// TwinCAT 3 PLC project Pecom_Drive_Communication
// Title: DCOS PecomDriveCommunication
// Company: DCOS
// Author: DCOS
// ProjectVersion: 1.0.0
// Description: Function for Drive Communication to manroland presses replacing Baumueller Drive systems
// ProgramVersion: 3.1.4024.0
// libraries:
//   Tc2_Standard, * (Beckhoff Automation GmbH)
//   Tc2_System, * (Beckhoff Automation GmbH)
//   Tc2_TcpIp, * (Beckhoff Automation GmbH)
//   Tc2_Utilities, * (Beckhoff Automation GmbH)
// project tree:
//   DUTs/DriveInterface/ ST_DriveInterface.TcDUT, ST_DriveInterface_Ctrl.TcDUT, ST_DriveInterface_Stat.TcDUT
//   DUTs/MainAxis_Interface/ ST_MainAxisInterface_Ctrl.TcDUT, ST_MainAxisInterface_Stat.TcDUT, ST_MainAxisInterface.TcDUT
//   DUTs/Pecom_Interface/Ethernet_TCP/ NETWORK_BUFFER.TcDUT, ST_ApplicationBinaryData.TcDUT, ST_BinaryFrame.TcDUT, ST_BinaryHeader.TcDUT, ST_TCP_Puff.TcDUT
//   DUTs/Pecom_Interface/Pecom_TCP/ ST_CommunicationStatus.TcDUT, ST_Elements.TcDUT, ST_InOut_Msg.TcDUT, ST_InOut_Data.TcDUT, ST_MsgBuffer.TcDUT, ST_Restart.TcDUT, ST_Objekt.TcDUT, ST_MemberAnounce.TcDUT
//   DUTs/Pecom_Interface/Pecom_UDP/ IP_C.TcDUT, ST_UDP_Buffer.TcDUT, ST_UDP_Drive_Data.TcDUT, ST_UDP_Msg_In.TcDUT, ST_UDP_Msg_Out.TcDUT
//   DUTs/Pecom_Interface/Setup_DriveCom/ ST_SetupDriveCom.TcDUT, ST_SetupDriveComMDS.TcDUT
//   DUTs/ ST_Alarm.TcDUT, ST_TCP_Parameter.TcDUT (not stored)
//   Global Variables/Pecom_Interface/ GVL_ConnectionAlarms.TcGVL, GVL_FB.TcGVL, GVL_Pecom.TcGVL, GVL_Setup.TcGVL, TCPIP_Constants.TcGVL
//   POUs/Network Functions/TCPIP_Communication/ FB_Server.TcPOU, FB_ServerApplication.TcPOU, FB_ServerConnection.TcPOU
//   POUs/Network Functions/TCPIP_Communication/Helper POUs/ FB_FrameFifo.TcPOU, FB_LogFifo.TcPOU, F_ADSLOGHEXDATA.TcPOU
//   POUs/Network Functions/UDP_Communication/ FB_UDP_Server.TcPOU, FB_UDP_Server_RESET.TcPOU
//   POUs/Pecom Interface/ PB_Start_TCPIP.TcPOU, PB_Start_UDP.TcPOU
//   POUs/Pecom Interface/Pecom_Functions/TCP Msg Handling/ Eth_Send_Receive.TcPOU, FB_Msg_Receive.TcPOU, FB_Msg_Send.TcPOU, FB_SendReceive_TcpIp.TcPOU, Pecom_In_Out_data.TcPOU, Trigger.TcPOU
//   POUs/Pecom Interface/Pecom_Functions/ Pecom_DriveMessage.TcPOU, Pecom_Write_Alarm.TcPOU
//   POUs/Pecom Interface/Pecom_Functions/UDP Msg Handling/ FB_UDP_DriveCom.TcPOU
//   POUs/UDFB/ DWORD_OF_BYTE.TcPOU, FC_Time_To_Ramp.TcPOU, WORD_OF_BYTE.TcPOU

// ---- DUTs/DriveInterface/ST_DriveInterface.TcDUT
TYPE ST_DriveInterface :
STRUCT
	stDriveMotorInterface_stat		: ST_DriveInterface_Stat;
	stDriveMotorInterface_ctrl		: ST_DriveInterface_Ctrl;
END_STRUCT
END_TYPE

// ---- DUTs/DriveInterface/ST_DriveInterface_Ctrl.TcDUT
TYPE ST_DriveInterface_Ctrl :
STRUCT
	nSelectedMaster			:WORD;				// selected master
	nClutchedMaster			:WORD;				// clutched master
	nDriveGroup				:INT;				// Group of drives for Cutoff and Webup -> It is like the Webnumber the drive belongs to
	bReset					:BOOL;				// rising trig will reset if any fault is active
	bEnable					:BOOL;				// set to give power to motor
	bStartRun				:BOOL;				// set to start motor in slow run
	bRunRev					:BOOL;				// Direction -> set to run motor in rev direcition
	fVelocity				:LREAL;				// selected speed for slow run, if = 0 then use default vel
	fAcceleration			:LREAL;				// Acceleration in Local mode
	nGearRatio				:INT;				// For 3.Folder -> 2 or 1 ; For Paddlewheel 10000 or 20000 depends on Collect or straight!!
	// Cutoff and Speedgain
	fSyncValue				:LREAL;				// relative value to the master where motor will clutch into
	fGain					:LREAL;				// speed offset in % where such value can be used 1 = 1% faster
	
	// Positioning
	bPositionMode			:BOOL;				// POS-Mode -> set to goto a modulated positon
	bPosDirection			:BOOL;				// POS-Mode -> what direction to use when finding modulated position
	fModeModPos				:LREAL;				// POS-Mode -> selected position for modulated position 0.000 - 360.000	
	
	// 3.Folder Speed Curve
	n3Folder_Offset			:LREAL;				// 3.Folder -> Additional Cutoff offset for the 3.Folder (Fixed Value from Plc)
	n3Folder_Offset_Curve	:LREAL;				// 3.Folder -> Speed Curve Offset
	n3Folder_Degree_Curve	:LREAL;				// 3.Folder -> steepness of the speed curve
	
	// Sync Mode and Sync Speed
	bDriveSyncMode_FW		:BOOL;				// Sync Forward --> Syncronisation-Speed can be any speed 
	bDriveSyncMode_BW		:BOOL;				// Sync Backward --> Syncronisation-Speed must be < Machine speed exept N= 0 !!!
	bDriveSyncMode_SW		:BOOL;				// Sync Shortest way --> Syncronisation-Speed must be < Machine speed exept N= 0 !!!
	fSyncSpeed				:LREAL;				// set to desired sync offset speed Degree/sec for sync to Main Axis
	fSpeedCR_Permill		:LREAL;				// For PU only!! -> 100.0000 Promill OR 0.0400 Promill
	fSpeedCR_DegreeS		:LREAL;				// For Folder only!! -> 20,0000 Degree/sec OR 1,0000 Degree/sec
	fSpeedCutoff_Permill_Vari	:LREAL;				// set to desired sync offset speed Promill -> eg. 100.0000 Promill OR 0.2800 Promill
	fSpeedCutoff_Degree		:LREAL;				// set to desired sync offset speed Degree/sec 
	
	
	// Webtension Control Mode 
	nWebTc_Mode				:INT;				// WebTc	-> 11=off, 12=On  , 13=Tempor. Off
	fWebTc_SpeedGain		:LREAL;				// WebTc	-> Speedgain in manual mode in permill * 100 (eg 0.01‰ * 100)
	fWebTc_WebTension		:LREAL;				// WebTc	-> Webtension in N In Automode
	
	// something ??
	nSwitchPararmeter		:DINT;				// Switches between 2 parameter sets -> 0 or 1
	bDriveMode				:BOOL;				// 11 = position Ctrl, 13 = speed Ctrl, 14 = Tourque slave
END_STRUCT
END_TYPE

// ---- DUTs/DriveInterface/ST_DriveInterface_Stat.TcDUT
TYPE ST_DriveInterface_Stat :
STRUCT
	bEnabled			:BOOL;			// drive is under power
	
	fActVel				:LREAL;			// acutal vel, untis/s
	fActTorque			:LREAL;			// Actual Torque in %
	fTemp				:REAL;			// actual motor temp
	fI2T				:REAL;			// actual current overload accumulator in % when at 100% drive will trip  
	
	bZeroSpeed			:BOOL;			// motor at zerospeed (standstill)
	
	// Sync Feedback
	bInSync				:BOOL;			// Drive is in Sync with master Axis
	
	// Error Handling
	bError				:BOOL;			// has fault	
	nErrorCode			:DINT;			// error code	
	
	//Positioning Mode
    bAtModPos			:BOOL;			// set when in modulated position mode and at required pos	
	fActPos				:LREAL;			// actual modulated position, units
	fSyncPosDifference	:LREAL;			// Difference of the MainAxis to the local Position
	// Webtension Control Mode 
	fWebTc_SpeedGain	:LREAL;		// WebTc	-> Speedgain in manual mode in permill * 100 (eg 0.01‰ * 100)
	fWebTc_WebTension	:LREAL;		// WebTc	-> Webtension in N In Automode
	
	
	// divers
	bCoolingFanStarted	:BOOL;			// coolingfan running
	bBrakeReleased		:BOOL;			// breake is off
END_STRUCT
END_TYPE

// ---- DUTs/MainAxis_Interface/ST_MainAxisInterface_Ctrl.TcDUT
TYPE ST_MainAxisInterface_Ctrl :
STRUCT
	bReset					:BOOL;						// rising trig will reset if any fault is active
	
	bEnable					:BOOL;						// set to give power to motor
	bStartRun				:BOOL;						// set to start motor in slow run
	fVelocity				:LREAL;						// selected speed for slow run, if = 0 then use default vel
	fAcceleration			:LREAL;						// Acceleration in Local mode
	
	// Cutoff and Speedgain
	fCutoffValue			:ARRAY[0..31] OF LREAL;		// Cutoff for each DriveGroup (equals the web number )
	
	// Aray of Cutoff values for each group
	aGroup_Cutoff			:	ARRAY[0..15] OF LREAL;	// Cutoff from SKS for each web Group
	
	// Each Bit represents a group which is doing a webbing up. Only drives in this group are turning
	aGroup_WebUpDrives		:	ARRAY[0..15] OF BOOL;	// Group which is involved in a webup			
	
END_STRUCT
END_TYPE

// ---- DUTs/MainAxis_Interface/ST_MainAxisInterface_Stat.TcDUT
TYPE ST_MainAxisInterface_Stat :
STRUCT
	bEnabled			:BOOL;			// drive is under power
	
	fActVel				:LREAL;			// acutal vel, untis/s
	
	fActPos				:LREAL;			// actual modulated position, units
	
	// P1160 Sync Feedback for each Drive Group (Bit 0 = Group 0 and so on)
	bInSync				:WORD;			// Status of the Sync Position for each DRIVE-GROUP (Is a drive in a group not in sync -> BIT is High)
	
	bZeroSpeed			:BOOL;			// motor at zerospeed (standstill)
	
	// Error Handling
	bError				:BOOL;			// Main Axis has a fault	


END_STRUCT
END_TYPE

// ---- DUTs/MainAxis_Interface/ST_MainAxisInterface.TcDUT
TYPE ST_MainAxisInterface :
STRUCT
	stMainAxisInterface_stat		: ST_MainAxisInterface_Stat;
	stMainAxisInterface_ctrl		: ST_MainAxisInterface_Ctrl;
END_STRUCT
END_TYPE

// ---- DUTs/Pecom_Interface/Ethernet_TCP/NETWORK_BUFFER.TcDUT
TYPE NETWORK_BUFFER :
STRUCT
	SIZE : UINT;
	BUFFER : ARRAY[0..Pecom_TCP_Puffer_Size] OF BYTE;
END_STRUCT
END_TYPE

// ---- DUTs/Pecom_Interface/Ethernet_TCP/ST_ApplicationBinaryData.TcDUT
(* Simple binary user data (8 byte aligned) *)
TYPE ST_ApplicationBinaryData :
STRUCT
	aData		: ARRAY[0..Pecom_TCP_Puffer_Size] OF BYTE; // 700 Byte
	reserved	: ARRAY[0..2] OF BYTE;(* Alignment data: 3 byte *)

END_STRUCT
END_TYPE

// ---- DUTs/Pecom_Interface/Ethernet_TCP/ST_BinaryFrame.TcDUT
(* Simple binary TCP/IP frame (8 byte aligned) *)
TYPE ST_BinaryFrame :
STRUCT
//	head	: ST_BinaryHeader;(* Frame header (16 byte) *)
	data 	: ST_ApplicationBinaryData;(* User data (120 byte) *)

	(* Total frame size = 136 byte *)
END_STRUCT
END_TYPE

// ---- DUTs/Pecom_Interface/Ethernet_TCP/ST_BinaryHeader.TcDUT
(* Simple binary TCP/IP frame header (8 byte aligned) *)
TYPE ST_BinaryHeader :
STRUCT
	dwStart		: DWORD	:= 16#BECF1234;	(* Start bytes *)
	cbLength	: UDINT(0..PLCPRJ_BUFFER_SIZE) := 0;(* Max. length of attached binary data *)
	nS			: UDINT := 0;(* Send counter *)
	nR			: UDINT	:= 0;(* Receive counter *)
	
	(* Total header data size = 16 byte *)
END_STRUCT
END_TYPE

// ---- DUTs/Pecom_Interface/Ethernet_TCP/ST_TCP_Puff.TcDUT
TYPE ST_TCP_Puff:
STRUCT
	Conected	: BOOL;
	Ip_Adresss	: T_IPv4addr;
	PecomTNR  	: INT;		 
	R_Buf		: NETWORK_BUFFER;
	S_Buf		: NETWORK_BUFFER;
END_STRUCT
END_TYPE

// ---- DUTs/Pecom_Interface/Pecom_TCP/ST_CommunicationStatus.TcDUT
TYPE ST_CommunicationStatus :
STRUCT
	stRestart				:	ST_Restart;
	bTCP_Connect			:	ARRAY[0..NR_OF_DRIVEMASTERS] OF BOOL;
	bUDP_Connect			:	ARRAY[0..NR_OF_DRIVEMASTERS] OF BOOL;
END_STRUCT
END_TYPE

// ---- DUTs/Pecom_Interface/Pecom_TCP/ST_Elements.TcDUT
TYPE ST_Elements :
STRUCT
	Nummer	  : INT;	(* Gegenstelle*)
	KNG	   	  : INT;
	ANFTYP	  : INT;
	SNSTIV	  : INT;
	ZYKTME	  : INT;
	MASEIN	  : INT;
	flag	  : BOOL;
END_STRUCT
END_TYPE

// ---- DUTs/Pecom_Interface/Pecom_TCP/ST_InOut_Msg.TcDUT
TYPE ST_InOut_Msg :
STRUCT
	number_of_buffers	:	INT;
	buffer_overfow		:	BOOL;
	Pecom_Tnr			:	ARRAY [1..40] OF INT;
	valid				:	ARRAY [1..40] OF BOOL;
	stMsgBuffer			:	ARRAY [1..40] OF  ST_MsgBuffer;	// 40 x 950 Words Buffer
END_STRUCT

END_TYPE

// ---- DUTs/Pecom_Interface/Pecom_TCP/ST_InOut_Data.TcDUT
TYPE ST_InOut_Data :
STRUCT
	Error						: SINT;
	Hand_Shake					: SINT;
    Receiver  					: INT;
	Sender     					: INT;
	Typ		 					: INT;
	NFB		  					: INT;
	Lg_Byte	 					: INT;
	KDO							: INT;
   	data						: ARRAY[7..950] OF INT;
	data_Max  					: INT;
   	BLK_Pointer 				: INT;
	DSK_Pointer 				: INT;
	nNumber_of_messages			: INT;
	nNumber_of_Error			: INT;
	nUnknown_message			: INT;
    data_transfer_ready     	: BOOL;
	data_are_valid				: BOOL;
	Send_data					: BOOL;
    job_running             	: BOOL;
	job_done 					: BOOL;
	job_not_done  				: BOOL;
	job_timeout					: BOOL;
	Release_first_value			: BOOL;
END_STRUCT
END_TYPE

// ---- DUTs/Pecom_Interface/Pecom_TCP/ST_MsgBuffer.TcDUT
(* Ethernetpuffer *)
TYPE ST_MsgBuffer :
STRUCT
	MSG	: ARRAY [0..950] OF	 WORD;	// Ethernetpuffer 950 Words
END_STRUCT
END_TYPE

// ---- DUTs/Pecom_Interface/Pecom_TCP/ST_Restart.TcDUT
TYPE ST_Restart :
STRUCT
	akt							: BOOL;
	TLN							: ARRAY[1..4]	OF	INT;
END_STRUCT
END_TYPE

// ---- DUTs/Pecom_Interface/Pecom_TCP/ST_Objekt.TcDUT
TYPE ST_Objekt :
STRUCT
    OBJART	  		: INT;
	OBJLGE	  		: INT;
	OBJGRP	  		: INT;
	OBJEIN	  		: INT;
	OBJLFN	  		: INT;
    AUFTRAG	  		: INT;
	KOM_RCK   		: BOOL;
	AKTIV			: BOOL;
	TLN				: ARRAY [0..4] OF ST_Elements;
	Read_Data 		: BOOL;
	Send_Data 		: BOOL;
	In_data			: ARRAY [0..400] OF INT;
	Out_data		: ARRAY [0..400] OF INT;

END_STRUCT
END_TYPE

// ---- DUTs/Pecom_Interface/Pecom_TCP/ST_MemberAnounce.TcDUT
TYPE ST_MemberAnounce :
STRUCT
	Laenge		:	WORD;
	receiver	:	WORD;
	Sender		:	WORD;
	Typ			:	WORD;
	Reserve		:	WORD;
	N_Laenge	:	WORD;
	Kommando	:	WORD;
END_STRUCT

END_TYPE

// ---- DUTs/Pecom_Interface/Pecom_UDP/IP_C.TcDUT
TYPE IP_C :
STRUCT
	C_PORT : WORD;						(*W Portnummer                                               *)
	C_IP : DWORD;						(*W IP-Adresse gepackt wwxxyyzz = www.xxx.yyy.zzz            *)
	C_STATE : BYTE;						(*R Verbindungsstatus ON/OFF + Flanke ON/OFF                 *)
	C_ENABLE : BOOL;					(*W Freigabe für Connect                                     *)
	R_OBSERVE : BOOL;					(*W Empfang ueberwachen                                      *)
	TIME_RESET : BOOL;					(*W Alle Timer ruecksetzen                                   *)
	ERROR : DWORD;					    (*R vvwwxxyy (vv = CON_ERROR, ww = SEN_ERROR, xx = REC_ERROR *)
	MAILBOX : ARRAY [1..16] OF BYTE;	(*I Mailbox: Datenbereich für Bausteindatenaustausch         *)
END_STRUCT
END_TYPE

// ---- DUTs/Pecom_Interface/Pecom_UDP/ST_UDP_Buffer.TcDUT
TYPE ST_UDP_Buffer :
STRUCT	
	Ip_Adresss		: T_IPv4addr;
	nDriveMemberNr	: INT;
	nPLCMemberNr	: INT;
	SIZE 			: UINT;
	BUFFER 			: ARRAY[0..Pecom_TCP_Puffer_Size] OF BYTE;
END_STRUCT
END_TYPE

// ---- DUTs/Pecom_Interface/Pecom_UDP/ST_UDP_Drive_Data.TcDUT
TYPE ST_UDP_Drive_Data :
	STRUCT
		sRemote_IP_Adress		: T_IPv4Addr;
		nDriveMemberNr			: INT;			// Own Pecom Member Nr. (Old MDS Pecom Nr)
		nPLCMemberNr			: INT;			// PLC Pecom Member Nr.
		bConnectionState		: BOOL;
		aDriveData_In			: ARRAY[0..50] OF ST_UDP_Msg_In;
		aDriveData_Out			: ARRAY[0..50] OF ST_UDP_Msg_Out;
	END_STRUCT
END_TYPE

// ---- DUTs/Pecom_Interface/Pecom_UDP/ST_UDP_Msg_In.TcDUT
TYPE ST_UDP_Msg_In :
	STRUCT
		nDriveSercos_Id			:	INT;
		nControlword			:	WORD;
		nSetpoint_speed			:	INT;	// Speed in Rev/10
		nSetpoint_Acceleration	:	INT;	// Acceleration /10 (Time in relation to Vmax eg. 37500 rev/h)
		bHandShake				:	BOOL;	// UDP Bit 0 Handshake
		bSyncRunMode			:	BOOL;	// UDP Bit 8 Syncron Run Operating Mode
		bPositionMode			:	BOOL;	// UDP Bit 9 Positioning Operating Mode
		bDriveEnable			:	BOOL;	// UDP Bit 14 Drive Enable
		bDriveStop				:	BOOL;	// UDP Bit 15 Drive Stop -> Drive is locked
	END_STRUCT
END_TYPE

// ---- DUTs/Pecom_Interface/Pecom_UDP/ST_UDP_Msg_Out.TcDUT
TYPE ST_UDP_Msg_Out :
	STRUCT
		nDriveSercos_Id			:	INT;
		nStatusWord				:	WORD;
		nActual_speed			:	INT;	// Actual Speed in Rev/10
		nActual_torque			:	INT;	// Torque in %
		bHandShake				:	BOOL;	// UDP Bit 0 Handshake
		bInSync					:	BOOL;	// UDP Bit 6 Drive in Sync
		bCommandDone			:	BOOL;	// UDP Bit 7 the last Command is executed
		bDriveFault				:	BOOL;	// UDP Bit 13 Drive has a fault
		bDriveActive			:	BOOL;	// UDP Bit 14 Drive is active (Enabled and run)
		bDriveReady				:	BOOL;	// UDP Bit 15 Drive is ready
	END_STRUCT
END_TYPE

// ---- DUTs/Pecom_Interface/Setup_DriveCom/ST_SetupDriveCom.TcDUT
TYPE ST_SetupDriveCom :
	STRUCT
		nDriveNumber			: INT;			// MDxx -> Drive number in the drive array and the Axis
		sDriveName				: STRING;		// Label of the drive eg. in the drawings
		sDriveDescription		: STRING;		// Description or function of the drive	in the press	
		sLocalIP				: STRING;		// Own Ip adress (Socket) where the Pecom send the Messages to
		sRemoteIP				: STRING;		// Ip adress of the pecom Partner-plc system 
		nDriveMemberNr			: INT;
		nPLCMemberNr			: INT;
        nSercosID               : INT;			// Indicate the position of the drive in the UDP-Msg Stack
	END_STRUCT
END_TYPE

// ---- DUTs/Pecom_Interface/Setup_DriveCom/ST_SetupDriveComMDS.TcDUT
TYPE ST_SetupDriveComMDS :
	STRUCT
		nUnitNr					: INT;
		stSetup_MDS_IP			: T_IPv4addr;
		nPLCMemberNr_1			: INT;
		nPLCMemberNr_2			: INT;
		nDriveMemberNr			: INT;
	END_STRUCT
END_TYPE

// ---- DUTs/ST_Alarm.TcDUT
TYPE ST_Alarm :
STRUCT
		Status				:	BOOL;
		ernr				:	INT;
		objektnr			:	INT;
		ort1				:	INT;
		ort2				:	INT;
		ort3				:	INT;
		ort4				:	INT;
		ort5				:	INT;
		ort6				:	INT;
		ort7				:	INT;
		ort8				:	INT;
		quitt				:	INT;
		sperre				:	INT;
		gruppe				:	INT;
END_STRUCT
END_TYPE

// ---- Global Variables/Pecom_Interface/GVL_ConnectionAlarms.TcGVL
VAR_GLOBAL
	bAlarm_NoUDP_Connection		:	ARRAY[0..NR_OF_DRIVEMASTERS] OF BOOL;
	bAlarm_NoTCP_Connection		:	ARRAY[0..NR_OF_DRIVEMASTERS] OF BOOL;

END_VAR

// ---- Global Variables/Pecom_Interface/GVL_FB.TcGVL
VAR_GLOBAL
	FB_UDP_Connection_arr	: ARRAY[0..NR_OF_DRIVEMASTERS] OF FB_UDP_DriveCom;
END_VAR

// ---- Global Variables/Pecom_Interface/GVL_Pecom.TcGVL
VAR_GLOBAL
	
	stDrive_Data_arr		:	ARRAY[0..NR_OF_DRIVEMASTERS]	OF ST_UDP_Drive_Data;
	aTcpPuff				:   ARRAY[0..NR_OF_DRIVEMASTERS] 	OF ST_TCP_Puff;
	UDP_SERVER_RESET 		: 	BYTE; 			// Set to 0 to close and reopen the UPD Socket (use R_TRIG !!) OK-State is 2
	
	stComStatus				:	ST_CommunicationStatus;
	(* PECOM messages *)
	st_IN_PecomMsg			:	ST_InOut_Msg;		// The TCP IN Buffer "R_BUF_A.BUFFER[x]" is copied into this Buffer
	st_OUT_PecomMsg			:	ST_InOut_Msg;		// This Buffer is transfered into the TCP Out Buffer -> "S_BUF_A.BUFFER[x]"
	st_IN_Objects			:	ST_InOut_Data;		// "st_IN_PecomMsg" are sorted into st_IN_Objects
	st_OUT_Objects			:	ST_InOut_Data;		// single "st_OUT_Objects" are sorted into "st_OUT_Objects_Buffer" and this finally into "st_OUT_PecomMsg"
	st_OUT_Objects_Buffer	:	ST_InOut_Data;		// "st_OUT_Objects_Buffer" transfered into "st_OUT_PecomMsg"
	st_OUT_Alarms			:	ST_InOut_Data;		// struct for Alarm Messages
	st_OUT_Alarms_Buffer	:	ST_InOut_Data;		// struct Buffer for Alarm Messages

END_VAR

// ---- Global Variables/Pecom_Interface/GVL_Setup.TcGVL
VAR_GLOBAL	
	stSetup_MdsCom				: ARRAY [0..NR_OF_DRIVEMASTERS] OF ST_SetupDriveComMDS;		
	stSetup_DriveCom			: ARRAY [0..50] 				OF ST_SetupDriveCom;
END_VAR

// ---- Global Variables/Pecom_Interface/TCPIP_Constants.TcGVL
VAR_GLOBAL CONSTANT
	
	NR_OF_DRIVEMASTERS						: USINT	:= 11;		(* Max. Number of TCP Connection and Server Instances *)

	Pecom_TCP_Puffer_Size					: INT	:= 700;	(* Puffer for the Pecom In/Out Messages *)
	PLCPRJ_BUFFER_SIZE						: UDINT := 1000;(* Max. internal fifo/receiver buffer size *)

(*	PLCPRJ_CLIENT_SEND_CYCLE_TIME			: TIME := T#1S; not used at server side *)
	PLCPRJ_RECEIVE_POLLING_TIME				: TIME := T#100MS;
	PLCPRJ_RECEIVE_TIMEOUT					: TIME := T#50S;

	(* Some project specific error codes *)
	PLCPRJ_ERROR_RECEIVE_TIMEOUT			: UDINT := 16#8101;(* Receive timeout *)
	PLCPRJ_ERROR_SENDFIFO_OVERFLOW			: UDINT := 16#8102;(* Send fifo overflow *)
	PLCPRJ_ERROR_RECFIFO_OVERFLOW			: UDINT := 16#8103;(* Receive fifo overflow *)
	PLCPRJ_ERROR_INVALID_FRAME_FORMAT		: UDINT := 16#8104;(* Invalid frame format/data *)
	
END_VAR

// ---- POUs/Pecom Interface/Pecom_Functions/UDP Msg Handling/FB_UDP_DriveCom.TcPOU
FUNCTION_BLOCK FB_UDP_DriveCom
VAR_INPUT
	sRemote_IP			: T_IPv4Addr;
	nDriveMemberNr		: INT;			// Own Pecom Member Nr. (Old MDS Nr)
	nPLCMemberNr		: INT;			// PLC Pecom Member Nr.
	p_UDP_DriveData		: POINTER TO ST_UDP_Drive_Data;
	S_BUF				: POINTER TO ST_UDP_Buffer;		// UDP Send Buffer It is hand over to the UDP Socket 
	R_BUF				: POINTER TO ST_UDP_Buffer;		// UDP Receive Buffer It comes from the UDP Socket 	

END_VAR
VAR_OUTPUT
	bAlarmNoConnection	: BOOL;
END_VAR

VAR
	nInPackageCount			: INT;
	bTimeout				: BOOL;
	TON_Timeout				: TON;
	nStackPointer			: INT;
	nDriveNumber			: INT;
	
	TO_PECOM				: ARRAY[0..650]	OF	WORD;
	TO_PECOM_old			: ARRAY[0..650]	OF	WORD;
	
	
	bSendRequest			: BOOL;
	nMsgSize				: INT;
	p						: INT;
	i						: INT;
	k						: UINT;
	sIPTEST: STRING(15);
END_VAR

(************************************************************************************************)
(*****				 					Ethernet UDP 										*****)
(***** UDP Communication between the PLC <--> Drive System 									*****)
(***** 																						*****)
(************************************************************************************************)
(*****			Time out or no connection after 7s of no Message		*****)
//Set the Timeout for connection control
bTimeout	:=	TRUE;
// Reset the TimeOut when you received a valid UDP-package
IF (R_BUF^.SIZE > 0 AND R_BUF^.Ip_Adresss = sRemote_IP) 
THEN
	bTimeout := FALSE;	
	nInPackageCount	:=	nInPackageCount	+	1;		// Diagnose Only!!
	sIPTEST	:= R_BUF^.Ip_Adresss;
END_IF
TON_Timeout(IN:= bTimeout, PT:=T#6S);
bAlarmNoConnection	:=	TON_Timeout.Q;

// Connection Flag in the UDP Buffer
p_UDP_DriveData^.bConnectionState := NOT bAlarmNoConnection	;

(****************************************************************************************)
(***							Receive Messages									*****)
(* If In-Buffer size is gt the 0 transfer the content to the  p_DriveData array			*)
(* In 1 Msg can be max. 48 drives controlled. Each on is identified by its Sercos-Id	*)
(****************************************************************************************)

IF		(R_BUF^.SIZE > 0 AND R_BUF^.Ip_Adresss = sRemote_IP)
THEN	
	p_UDP_DriveData^.sRemote_IP_Adress	:= 	sRemote_IP;
	p_UDP_DriveData^.nDriveMemberNr		:=	R_BUF^.nDriveMemberNr;	
	p_UDP_DriveData^.nPLCMemberNr		:=	R_BUF^.nPLCMemberNr;
	nStackPointer	:=	26;	// Pointer offset to the First drive information in the Msg
	
	FOR nDriveNumber	:= 0 TO 48
				DO
					p_UDP_DriveData^.aDriveData_In[nDriveNumber].nDriveSercos_Id		:=	WORD_TO_INT(WORD_OF_BYTE(R_BUF^.BUFFER[nStackPointer+1],R_BUF^.BUFFER[nStackPointer]));
					p_UDP_DriveData^.aDriveData_In[nDriveNumber].nControlword 			:=	WORD_OF_BYTE(R_BUF^.BUFFER[nStackPointer+2],R_BUF^.BUFFER[nStackPointer+3]);
					p_UDP_DriveData^.aDriveData_In[nDriveNumber].nSetpoint_speed 		:=	WORD_TO_INT(WORD_OF_BYTE(R_BUF^.BUFFER[nStackPointer+4],R_BUF^.BUFFER[nStackPointer+5]));
					p_UDP_DriveData^.aDriveData_In[nDriveNumber].nSetpoint_Acceleration :=	WORD_TO_INT(WORD_OF_BYTE(R_BUF^.BUFFER[nStackPointer+6],R_BUF^.BUFFER[nStackPointer+7]));
					
					// Assign the Control bits
					p_UDP_DriveData^.aDriveData_In[nDriveNumber].bHandShake				:=	p_UDP_DriveData^.aDriveData_In[nDriveNumber].nControlword.0;
					p_UDP_DriveData^.aDriveData_In[nDriveNumber].bSyncRunMode			:=	p_UDP_DriveData^.aDriveData_In[nDriveNumber].nControlword.8;
					p_UDP_DriveData^.aDriveData_In[nDriveNumber].bPositionMode			:=	p_UDP_DriveData^.aDriveData_In[nDriveNumber].nControlword.9;
					p_UDP_DriveData^.aDriveData_In[nDriveNumber].bDriveEnable			:=	p_UDP_DriveData^.aDriveData_In[nDriveNumber].nControlword.14;
					p_UDP_DriveData^.aDriveData_In[nDriveNumber].bDriveStop				:=	p_UDP_DriveData^.aDriveData_In[nDriveNumber].nControlword.15;

					nStackPointer	:= nStackPointer +12;
	END_FOR;		
END_IF

(****************************************************************************************)
(***							Send Messages									*****)
(* If In-Buffer size is gt the 0 transfer the content to the  p_DriveData array			*)
(* In 1 Msg can be max. 48 drives controlled. Each on is identified by its Sercos-Id	*)
(****************************************************************************************)
TO_PECOM_old := TO_PECOM;
(*****************************************************)
(** Build the Header of the Message					**)
(**	static part of the message 						**)
(*****************************************************)

TO_PECOM[0]		:=	INT_TO_WORD(nPLCMemberNr);
TO_PECOM[1]		:=	INT_TO_WORD(nDriveMemberNr);
TO_PECOM[2]		:=	WORD#153;
TO_PECOM[3]		:=	WORD#0;
TO_PECOM[4]		:=	WORD#600;	(* 12 Byte x 49 Drives *)
TO_PECOM[5]		:=	WORD#10912;	(* Message Type	*)
TO_PECOM[6]		:=	WORD#0;
TO_PECOM[7]		:=	WORD#1;
TO_PECOM[8]		:=	WORD#302;	(* OBJART *)
TO_PECOM[9]		:=	WORD#49;	(* number of drives *)
TO_PECOM[10]	:=	WORD#12;	(* OBJLGE per Drive in Byte*)


(*****************************************************)
(**	dynamic part of the message 					**)
(*****************************************************)
// Write the Drive struct into the temp. Send-Buffer
p	:=	11;
	FOR nDriveNumber	:= 0 TO 48
		DO	p_UDP_DriveData^.aDriveData_Out[nDriveNumber].nStatusWord	:= 0;	// Clear the Status
		
			// reply to the UDP Handshake Bit
			p_UDP_DriveData^.aDriveData_Out[nDriveNumber].bHandShake		:= p_UDP_DriveData^.aDriveData_In[nDriveNumber].bHandShake;

			// Write the Status word
			p_UDP_DriveData^.aDriveData_Out[nDriveNumber].nStatusWord.0		:= p_UDP_DriveData^.aDriveData_Out[nDriveNumber].bHandShake;
			p_UDP_DriveData^.aDriveData_Out[nDriveNumber].nStatusWord.6		:= p_UDP_DriveData^.aDriveData_Out[nDriveNumber].bInSync;
			p_UDP_DriveData^.aDriveData_Out[nDriveNumber].nStatusWord.7		:= p_UDP_DriveData^.aDriveData_Out[nDriveNumber].bCommandDone;
			p_UDP_DriveData^.aDriveData_Out[nDriveNumber].nStatusWord.13	:= p_UDP_DriveData^.aDriveData_Out[nDriveNumber].bDriveFault;			
			p_UDP_DriveData^.aDriveData_Out[nDriveNumber].nStatusWord.14	:= p_UDP_DriveData^.aDriveData_Out[nDriveNumber].bDriveReady;
			p_UDP_DriveData^.aDriveData_Out[nDriveNumber].nStatusWord.15	:= p_UDP_DriveData^.aDriveData_Out[nDriveNumber].bDriveActive;
		
			TO_PECOM[p]		:=	2056;
			TO_PECOM[p+1]	:=	1;
			TO_PECOM[p+2]	:=	ROR(INT_TO_WORD(p_UDP_DriveData^.aDriveData_In[nDriveNumber].nDriveSercos_Id),8);
			TO_PECOM[p+3]	:=	p_UDP_DriveData^.aDriveData_Out[nDriveNumber].nStatusWord;
			TO_PECOM[p+4]	:=	INT_TO_WORD(p_UDP_DriveData^.aDriveData_Out[nDriveNumber].nActual_speed);
			TO_PECOM[p+5]	:=	INT_TO_WORD(p_UDP_DriveData^.aDriveData_Out[nDriveNumber].nActual_torque);
			nMsgSize		:=  p *2;
			p	:= p + 6;
			
END_FOR

(*****************************************************)
(***	Create a send request					******)
(*****************************************************)
// Compare old and new State and create a SendRequest

IF 	MEMCMP(ADR(TO_PECOM), ADR(TO_PECOM_old), SIZEOF(TO_PECOM_old)) <> 0	
	OR	(R_BUF^.SIZE > UINT#0 AND R_BUF^.Ip_Adresss = sRemote_IP)		(*message was incoming and must be replied*)
THEN
	bSendRequest:=	TRUE;
END_IF

(*****************************************************)
(* send the message to the remote plc*)
(*****************************************************)
IF bSendRequest THEN	
	IF	S_BUF^.SIZE	=	UINT#0 (* last message was done *)
	THEN
		k	:=	0;
		FOR	i	:= 0 TO nMsgSize
			DO
				S_BUF^.BUFFER[k]		:=	WORD_TO_BYTE(SHR(TO_PECOM[i],8));
				k	:=	k + 1;
				S_BUF^.BUFFER[k]		:=	WORD_TO_BYTE(TO_PECOM[i]);				
				k	:=	k + 1;
			END_FOR;
		S_BUF^.Ip_Adresss 				:= sRemote_IP;
		S_BUF^.nPLCMemberNr				:= nPLCMemberNr;
		S_BUF^.nDriveMemberNr			:= nDriveMemberNr;
		S_BUF^.SIZE						:= k;			(* send it *)
		bSendRequest 					:= FALSE;		
	END_IF;	
END_IF

(********************************************************)
(* Reset the Receiving buffer and wait for next message	*)
(*****************************************************)
IF R_BUF^.Ip_Adresss = sRemote_IP THEN
	R_BUF^.SIZE	:=	0;
	R_BUF^.Ip_Adresss := '';
END_IF

END_FUNCTION_BLOCK

// ---- POUs/UDFB/WORD_OF_BYTE.TcPOU
FUNCTION WORD_OF_BYTE : WORD
VAR_INPUT
	B1 : BYTE;
	B0 : BYTE;
END_VAR


(*
version 1.4	18. jul. 2009
programmer 	hugo
tested by		tobias

this function creates a word from 2 individual bytes

*)

WORD_OF_BYTE := SHL(BYTE_TO_WORD(B1),8) OR BYTE_TO_WORD(B0);

(* revision history
hm	24. jan 2007	rev 1.0
	original version

hm	2. jan 2008	rev 1.1
	improved performance

hm	19. feb 2008	rev 1.2
	replaced and with or for better compatibility

hm	23. apr. 2008	rev 1.3
	reverse order of inputs to be more logical

hm	18. jul. 2009	rev 1.4
	added type conversions for compatibility reasons

*)

END_FUNCTION

// ---- POUs/Network Functions/TCPIP_Communication/FB_Server.TcPOU
FUNCTION_BLOCK FB_Server
VAR_IN_OUT
	hServer			: T_HSERVER;(* Server connection handle *)
END_VAR
VAR_INPUT
	nServer_Id		: INT;
	sSrvNetID		: T_AmsNetID	:= '';(* TwinCAT TCP/IP server network address *)
	bEnable			: BOOL 			:= FALSE;(* TRUE => Enable server data exchange, FALSE => Disable *)
	bLog			: BOOL 			:= FALSE;(* TRUE => Enable log message output, FALSE => Disable *)
	sPrefix			: STRING 		:= 'SERVER::';(* Log message description string (allows the identification of log message source) *)
END_VAR
VAR_OUTPUT
	eState			: E_SocketConnectionState := eSOCKET_DISCONNECTED;(* TCP/IP connection state *)
END_VAR
VAR
	fbApplication 	: FB_ServerApplication;(* Server application control function block *)
	fbConnection	: FB_ServerConnection;(* Server data exchange control function block *)
	fbTx 			: FB_FrameFifo;(* Tx fifo *)
	fbRx 			: FB_FrameFifo;(* Rx fifo *)
	fbLog			: FB_LogFifo;(* Log/debug/error fifo *)
END_VAR

(*-------------------------- Trigger data exchange -----------------------------------------------*)
fbConnection( 	hServer := hServer, sSrvNetID := sSrvNetID, 
				fbRx := fbRx, fbTx := fbTx, fbLog := fbLog, 
				bEnable := bEnable, bLog := bLog, sPrefix := sPrefix, eState=>eState );
	
IF fbConnection.eState = eSOCKET_CONNECTED THEN(* Connection established *)
	aTcpPuff[nServer_Id].Conected := TRUE;
	aTcpPuff[nServer_Id].Ip_Adresss := fbConnection.sIpAdress;
	fbApplication( fbTx := fbTx, fbRx := fbRx, fbLog := fbLog, nServer_Id := nServer_Id );
ELSE	
	aTcpPuff[nServer_Id].Ip_Adresss := '';
	aTcpPuff[nServer_Id].PecomTNR 	:= 0;
	aTcpPuff[nServer_Id].Conected 	:= FALSE;
END_IF

END_FUNCTION_BLOCK

// ---- POUs/Network Functions/TCPIP_Communication/FB_ServerApplication.TcPOU
(* Sample server application. Adapt this code to match your needs. *)
FUNCTION_BLOCK FB_ServerApplication
VAR_INPUT	
	nServer_Id		: INT;
END_VAR
VAR_IN_OUT
	fbTx 			: FB_FrameFifo;(* TX fifo *)
	fbRx 			: FB_FrameFifo;(* RX fifo *)
	fbLog			: FB_LogFifo;(* Log message fifo *)
END_VAR
VAR
	stToClient		: ST_ApplicationBinaryData; (* Tx user data *)
	stFromClient	: ST_ApplicationBinaryData; (* Rx user data *)
	sLogMessage 	: T_MaxString := '';(* Log/debug/error message *)
END_VAR

(*------------------- Fetch rx data and send them back to the client -------------------------------------------------- *)
REPEAT
(*********************************************************************************************)	
(************************** Read DataFrom the Receive-Buffer	**********************************)
(*********************************************************************************************)	
	fbRx.RemoveHead( );(* Fetch data from rx fifo *)
	IF fbRx.bOk  THEN(* Success *)
		stFromClient := fbRx.stGet;				
		aTcpPuff[nServer_Id].R_Buf.BUFFER := stFromClient.aData;
		aTcpPuff[nServer_Id].R_Buf.SIZE	:= UDINT_TO_UINT(fbRx.nNrOfByteRead);		
	END_IF
	
(*********************************************************************************************)	
(************************** Write Data to the Send-Buffer	**********************************)
(*********************************************************************************************)	
	IF aTcpPuff[nServer_Id].S_Buf.SIZE > 0 THEN	
		stToClient.aData	:= 	aTcpPuff[nServer_Id].S_Buf.BUFFER;	
		fbTx.nSizeToWrite	:= aTcpPuff[nServer_Id].S_Buf.SIZE;	
		aTcpPuff[nServer_Id].S_Buf.SIZE := 0;	
		fbTx.AddTail( stPut := stToClient );(* Put user data to the tx fifo *)
		IF NOT fbTx.bOk THEN(* Fifo overflow => Log error *)
			fbLog.Error( sMessage := 'FB_FrameFifo(sender)', nErrID := PLCPRJ_ERROR_SENDFIFO_OVERFLOW );
		END_IF
	END_IF		
	
UNTIL NOT fbRx.bOk
END_REPEAT

(*---------------------- Get log/error messages from log fifo ------------------*)
REPEAT
	fbLog.Remove( );
	IF fbLog.bOk THEN

		(* TODO: Implement log message handler *)
		sLogMessage := fbLog.sGet;

	END_IF
UNTIL NOT fbLog.bOk
END_REPEAT

END_FUNCTION_BLOCK

// ---- POUs/Network Functions/TCPIP_Communication/Helper POUs/FB_FrameFifo.TcPOU
(* Tx/Rx (string data) fifo control function block *)
FUNCTION_BLOCK FB_FrameFifo
VAR_INPUT
	bLog		: BOOL		:= FALSE;		(* TRUE => Enable log message output, FALSE => Disable *)
	sPrefix		: STRING	:= 'Unknown::';	(* Log message description string (allows the identification of log message source) *)
	stPut		: ST_ApplicationBinaryData;	(* Frame to add (write) to the fifo *)
	nSizeToWrite: UDINT;					(* Size of Message to write *)
END_VAR
VAR_OUTPUT
	bOk			: BOOL; 					(* TRUE = New entry added or removed succesfully, FALSE = Fifo overflow or fifo empty *)
	stGet		: ST_ApplicationBinaryData;	(* Frame removed (read) from fifo *)
	nCount		: UDINT		:= 0;			(* Number of fifo entries *)
	cbFree		: UDINT 	:= 0;			(* Free buffer space *)
	nNrOfByteRead : UDINT;					(* Number of Byte read from the last Message received  *)
END_VAR
VAR
	fbBuffer 	: FB_MemRingBuffer;(* Basic (lower level) buffer control function block *)
	buffer		: ARRAY[-3..PLCPRJ_BUFFER_SIZE] OF BYTE;(* Internal buffer memory *)
END_VAR

;

ACTION AddTail:
(* Adds new fifo entry *)
fbBuffer.A_AddTail( pBuffer:= ADR(buffer), 			// Pointer to ring Buffer Data bytes
					cbBuffer:= SIZEOF(buffer),		// Maximum ring Puffer Size
					pWrite := ADR( stPut ), 		// Pointer to Write data
					cbWrite := nSizeToWrite, 	    // Buffersize of Write Data -> Must match the pecom message size!!
					bOk=>bOk,
					nCount=>nCount );									
					
IF bOk THEN
	cbFree := PLCPRJ_BUFFER_SIZE - fbBuffer.cbSize;(* Calculate the free buffer space *)
	IF bLog THEN(* Log message *)
		F_ADSLOGHEXDATA( CONCAT( sPrefix, '<=' ), ADR( stPut ), SIZEOF( stPut ) );
	END_IF
END_IF
END_ACTION

ACTION Clear:
(* Resets fifo = clears all data *)
MEMSET( ADR( stGet ), 0, SIZEOF( stGet ) );
fbBuffer.A_Reset( pBuffer:= ADR(buffer), cbBuffer:= SIZEOF(buffer),
					pWrite := ADR( stPut ), cbWrite := SIZEOF( stPut ), 
					pRead := ADR( stGet ), cbRead := SIZEOF( stPut ),
					bOk=>bOk, nCount=>nCount );
cbFree := PLCPRJ_BUFFER_SIZE;(* Free buffer size *)
END_ACTION

ACTION RemoveHead:
(* Removes oldest fifo entry *)
MEMSET( ADR( stGet ), 0, SIZEOF( stGet ) );
fbBuffer.A_RemoveHead( pBuffer:= ADR(buffer), cbBuffer:= SIZEOF(buffer),
						pRead := ADR( stGet ), cbRead := SIZEOF( stGet ),
						bOk=>bOk, nCount=>nCount );
IF bOk THEN
	nNrOfByteRead	:= fbBuffer.cbReturn;	// Return number of received Bytes
	cbFree 			:= PLCPRJ_BUFFER_SIZE - fbBuffer.cbSize;(* Calculate the free buffer space *)
END_IF
END_ACTION

END_FUNCTION_BLOCK

// ---- POUs/Network Functions/TCPIP_Communication/Helper POUs/F_ADSLOGHEXDATA.TcPOU
(* This function logs hexadecimal data to the TwinCAT XAE->Error list window *)
FUNCTION F_ADSLOGHEXDATA : DINT
VAR_INPUT
	sPrefix		: STRING;(* Debug message prefix string (allows the identification of log message source) *)
	pBuffer		: PVOID;(* Address of source buffer *)
	cbBuffer	: UDINT;(* Byte size of source buffer *)
END_VAR
VAR
	fbSplit	: FB_MemBufferSplit;
	sArg	: T_MaxString;
	sFormat : STRING;
END_VAR

IF pBuffer = 0 OR cbBuffer = 0 THEN
	RETURN;
END_IF

sFormat := CONCAT( sPrefix, '%s' );
fbSplit.eCmd := eEnumCmd_First;

REPEAT
	fbSplit( pBuffer := pBuffer, cbBuffer := cbBuffer, cbSize := 32 );(* Split binary data to 32 byte segments *)
	IF fbSplit.bOk THEN

		sArg := DATA_TO_HEXSTR( pData := fbSplit.pSegment, cbData := fbSplit.cbSegment, FALSE );(* Convert binary data to hex string *)

		F_ADSLOGHEXDATA := ADSLOGSTR( ADSLOG_MSGTYPE_HINT OR ADSLOG_MSGTYPE_LOG, sFormat, sArg );(* Log hex string *)

		sFormat := '%s';
		fbSplit.eCmd := eEnumCmd_Next;
	END_IF
UNTIL NOT fbSplit.bOk
END_REPEAT

END_FUNCTION

// ---- POUs/Network Functions/TCPIP_Communication/Helper POUs/FB_LogFifo.TcPOU
(* Log/debug/error message fifo *)
FUNCTION_BLOCK FB_LogFifo
VAR_INPUT
	bLog		: BOOL 		:= FALSE;(* TRUE => Enable log message output, FALSE => Disable *)
	sPrefix		: STRING 	:= 'Unknown::';(* Log message description string (allows the identification of log message source) *)
	
	sMessage	: STRING 	:= '';(* String message to add (write) to the fifo *)
	nErrID		: UDINT 	:= 0;(* Error code to add (write) to the fifo *)
	hSocket		: T_HSOCKET;(* Socket connection handle *)
END_VAR
VAR_OUTPUT
	bOk			: BOOL;(* TRUE = New entry added or removed succesfully, FALSE = Fifo overflow or fifo empty *)
	sGet		: T_MaxString := '';(* String entry removed (read) from fifo *)
	nCount		: UDINT := 0;(* Number of fifo entries *)
END_VAR
VAR
	fbBuffer 	: FB_StringRingBuffer;(* Basic (lower level) string buffer control function block *)
	buffer		: ARRAY[0..PLCPRJ_BUFFER_SIZE] OF BYTE;(* Internal buffer memory *)
	sSource		: T_MaxString;	
	sPut		: T_MaxString;
END_VAR

;

ACTION Clear:
(* Clears all fifo entries *)
fbBuffer.A_Reset( 	pBuffer := ADR( buffer ), cbBuffer := SIZEOF( buffer ), 
					bOk=>bOk, nCount=>nCount, getValue=>sGet );
END_ACTION

ACTION Error:
(* Adds new fifo entry *)
IF nErrID = 0 THEN
	sSource := '::Error: 0x';
ELSIF ( nErrID AND 16#80000000) = 16#80000000 THEN
	IF nErrID = 16#80072746 THEN
		sSource := '::Win32 error (the connection is reset by remote side): 0x';
	ELSE
		sSource := '::Win32 error: 0x';
	END_IF
ELSIF (nErrID AND 16#00008100) = 16#00008100 THEN
	CASE nErrID OF
		PLCPRJ_ERROR_RECEIVE_TIMEOUT:
			sSource := '::PLC sample project receive timeout error: 0x';
		PLCPRJ_ERROR_SENDFIFO_OVERFLOW:
			sSource := '::PLC sample project send fifo overflow error: 0x';
		PLCPRJ_ERROR_RECFIFO_OVERFLOW:
			sSource := '::PLC sample project receive fifo overflow error: 0x';
		PLCPRJ_ERROR_INVALID_FRAME_FORMAT:
			sSource := '::PLC sample project invalid frame format error: 0x';
	ELSE
		sSource := '::Other PLC sample project error: 0x';
	END_CASE
ELSIF (nErrID AND 16#00008000) = 16#00008000 THEN
	sSource := '::Internal TCP/IP Connection Server error: 0x';
ELSE
	sSource := '::TwinCAT System error: 0x';
END_IF

sPut := CONCAT( CONCAT( CONCAT( sPrefix, sMessage ), sSource ), DWORD_TO_HEXSTR( nErrID AND 16#FFFF, 0, FALSE ) ); 

fbBuffer.A_AddTail( pBuffer:= ADR(buffer), cbBuffer:= SIZEOF(buffer),
					putValue:= sPut, bOk=>bOk, nCount=>nCount );
IF bOk THEN
	IF bLog THEN(* Log error message *)
		ADSLOGSTR( ADSLOG_MSGTYPE_ERROR OR ADSLOG_MSGTYPE_LOG, '%s', sPut );	
	END_IF
END_IF
END_ACTION

ACTION Message:
(* Adds new fifo entry *)
sPut := CONCAT( CONCAT( sPrefix, sMessage ), CONCAT( '::', HSOCKET_TO_STRING(hSocket) ) );
fbBuffer.A_AddTail( pBuffer:= ADR(buffer), cbBuffer:= SIZEOF(buffer),
					putValue:= sPut, bOk=>bOk, nCount=>nCount );
IF bOk THEN
	IF bLog THEN(* Log information message *)
		ADSLOGSTR( ADSLOG_MSGTYPE_HINT OR ADSLOG_MSGTYPE_LOG, '%s', sPut );	
	END_IF
END_IF
END_ACTION

ACTION Remove:
(* Removes oldest fifo entry *)
IF nCount = 0 THEN
	sGet := '';
	bOk := FALSE;
	RETURN;
END_IF

fbBuffer.A_RemoveHead( pBuffer:= ADR(buffer), cbBuffer:= SIZEOF(buffer),
						getValue=>sGet, bOk=>bOk, nCount=>nCount );
END_ACTION

END_FUNCTION_BLOCK

// ---- POUs/Network Functions/TCPIP_Communication/FB_ServerConnection.TcPOU
(* 	This function block implements simple TCP/IP server protocol. *)
FUNCTION_BLOCK FB_ServerConnection
VAR_IN_OUT
	hServer		: T_HSERVER;(* Server connection handle *)
	fbTx 		: FB_FrameFifo;(* TX fifo *)
	fbRx 		: FB_FrameFifo;(* RX fifo *)
	fbLog		: FB_LogFifo;(* Log message fifo *)
END_VAR
VAR_INPUT
	sSrvNetID	: T_AmsNetID	:= '';(* TwinCAT TCP/IP server network address *)
	bEnable		: BOOL			:= FALSE;(* TRUE => Enable/connect, FALSE => Disable/disconnect *)
	tReconnect	: TIME 			:= T#1S;(* Try to reconnect after this time *)
	bLog		: BOOL 			:= FALSE; (* TRUE => Enable debug output, FALSE => Disable debug output *)
	sPrefix		: STRING 		:= 'SERVER::';(* Log message description string (allows the identification of log message source) *)
END_VAR
VAR_OUTPUT
	sIpAdress	: T_IPv4Addr;
	eState		: E_SocketConnectionState := eSOCKET_DISCONNECTED;(* TCP/IP connection state *)
END_VAR
VAR
	fbConnect 	: FB_ServerClientConnection;(* Create/release TCP/IP connection *)
	fbSend		: FB_SocketSend;(* Send TCP/IP data *)
	fbReceive	: FB_SocketReceive;(* Receive TCP/IP data *)
	nState 		: BYTE;(* Global state *)
	bSndBusy 	: BOOL;(* Tx state *)
	bRcvBusy 	: BOOL;(* Rx state *)
	bDisconnect	: BOOL;(* Disconnect flag, if set the socket will be closed *)

	fbPollTimer	: TON;(* Rx data poll timer *)
	fbRequestTimer	: TON;(* Request timeout timer *)
	fbReconnectTimer : TON;(* Reconnect timer *)

	nS			: UDINT;(* Send frame counter *)
	nR			: UDINT;(* Received frame counter *)
	cbReceived	: UDINT;(* Count of received data bytes *)
	rxBuffer	: ARRAY[0..PLCPRJ_BUFFER_SIZE] OF BYTE;
	cbFrame		: UDINT;(* Rx frame byte size *)
	stTxFrame	: ST_BinaryFrame;(* Tx frame buffer (inclusive header) *)
	stRxFrame	: ST_BinaryFrame;(* Rx frame buffer (inclusive header) *)
	bAbort		: BOOL;(* Flag to abort frame parsing loop *)
END_VAR

CASE nState OF
	0:(* Create TCP/IP connection *)
		fbConnect( 	eMode := eACCEPT_ALL, tReconnect := tReconnect, bEnable := bEnable, 
					hServer := hServer, eState => eState );
		IF NOT fbConnect.bBusy THEN
			IF NOT fbConnect.bError THEN
				IF eState = eSOCKET_CONNECTED THEN(* we are connected *)
					
					fbTx.Clear( sPrefix := CONCAT( sPrefix, 'FB_FrameFifo(sender)::' ), bLog := bLog );(* Clear TX fifo (optional) *)
					fbRx.Clear( sPrefix := CONCAT( sPrefix, 'FB_FrameFifo(receiver)::' ), bLog := bLog );(* Clear RX fifo (optional) *)
					fbLog.Clear( sPrefix := sPrefix, bLog := bLog );(* Clear log fifo (optional) *)
					bSndBusy := FALSE;
					bRcvBusy := FALSE;
					bDisconnect := FALSE;
					cbReceived 	:= 0;(* Reset number of received data bytes *)

					fbPollTimer( IN := FALSE, PT := T#0S );
					fbRequestTimer( IN := FALSE, PT := PLCPRJ_RECEIVE_TIMEOUT );
					fbReconnectTimer( IN := FALSE, PT := tReconnect );
				
					fbLog.Message( sMessage := 'Connection established!', hSocket := fbConnect.hSocket );
					nState 	:= 1;			
					sIpAdress:=fbConnect.hSocket.remoteAddr.sAddr;
				END_IF
			ELSE(* Connect error => log error *)
				fbLog.Error( sMessage := 'FB_ServerClientConnection()', nErrID := fbConnect.nErrId );
			END_IF
		END_IF


	1:(* Data exchange state *)
		bDisconnect := NOT bEnable OR bDisconnect;(* User/internal disconnect requested? *)
		IF bDisconnect AND NOT bSndBusy AND NOT bRcvBusy THEN
			bDisconnect := FALSE;
			fbLog.Message( sMessage := 'Closing connection!', hSocket := fbConnect.hSocket );
			nState := 2;(* Disconnect *)
		ELSE

			(* ----------------------- Get/fetch rx data -------------------------------- *)
			IF NOT bDisconnect AND NOT bRcvBusy THEN
				fbPollTimer( IN := TRUE );
				IF fbPollTimer.Q THEN
					IF fbRx.cbFree >= SIZEOF(stRxFrame.data) THEN(* Check free rx fifo space *)
						fbPollTimer( IN := FALSE, PT := PLCPRJ_RECEIVE_POLLING_TIME );
						fbReceive( bExecute := FALSE );
						fbReceive( 	sSrvNetId	:= sSrvNetID,
									hSocket		:= fbConnect.hSocket,
									cbLen		:= SIZEOF(stRxFrame),
									pDest		:= ADR(stRxFrame),
									bExecute	:= eState = eSOCKET_CONNECTED );
						bRcvBusy := eState = eSOCKET_CONNECTED;
					END_IF
				END_IF
				
			ELSE(* Wait until receive not busy *)
				
				fbReceive( bExecute := FALSE );
				IF NOT fbReceive.bBusy THEN
					bRcvBusy := FALSE;
					IF NOT fbReceive.bError THEN
						IF fbReceive.nRecBytes > 0 THEN (* Some bytes received *)

							fbPollTimer( IN := FALSE, PT := T#0S );(* Bytes received => increase the read (polling) speed *)
							cbReceived := fbReceive.nRecBytes;
							fbRx.AddTail( stPut := stRxFrame.data,nSizeToWrite := cbReceived);(* Add user data to the rx fifo *)
							IF fbRx.bOk THEN
								IF fbRx.cbFree >= SIZEOF(stRxFrame.data) THEN
									bAbort := FALSE;(* reset flag, try to parse next frame *)
								END_IF
							ELSE (* Fifo overflow => log error and disconnect *)
								fbLog.Error( sMessage := 'FB_FrameFifo(receiver)', nErrID := PLCPRJ_ERROR_RECFIFO_OVERFLOW );
								bDisconnect := TRUE;(* Set flag *)
								RETURN;
							END_IF		
						END_IF

					ELSE(* Receive error => Log error and disconnect *)
						fbLog.Error( sMessage := 'FB_SocketReceive()', nErrID := fbReceive.nErrId );
						bDisconnect := TRUE;(* set flag *)
					END_IF

				END_IF(* IF NOT fbReceive.bBusy THEN *)
				
			END_IF(* IF NOT bDisconnect AND NOT bRcvBusy THEN *)
			(* -------------------------------------------------------------------------- *)

			
			
			(* ------------------------------ Send tx data ------------------------------ *)
			IF NOT bDisconnect AND NOT bSndBusy THEN
				fbTx.RemoveHead();(* Remove oldest user data entry *)
				IF fbTx.bOk THEN(* Success *)
						
					stTxFrame.data := fbTx.stGet;
					fbTx.nSizeToWrite;			
					(* Send frame *)
					fbSend( bExecute := FALSE );
					fbSend(	sSrvNetID 	:= sSrvNetID,
							hSocket		:= fbConnect.hSocket,
							cbLen		:= fbTx.nSizeToWrite,	(* size of user data *)
							pSrc		:= ADR(stTxFrame),(* Pointer to the frame data *)
							bExecute	:= TRUE );
					bSndBusy := TRUE;
				END_IF
			ELSE(* Wait until send not busy *)
				fbSend( bExecute := FALSE );
				IF NOT fbSend.bBusy THEN
					bSndBusy := FALSE;
					IF NOT fbSend.bError THEN(* No error *)
					ELSE(* Send error => Log error and disconnect *)
						fbLog.Error( sMessage := 'FB_SocketSend()', nErrID := fbSend.nErrId );
						bDisconnect := TRUE;(* Set flag *)
					END_IF
				END_IF
			END_IF
			(* -------------------------------------------------------------------------- *)

			
		END_IF(* IF bDisconnect AND NOT bSndBusy AND NOT bRcvBusy THEN *)


	2:(* Disconnect *)
		fbConnect( hServer := hServer, bEnable:= FALSE, eState=>eState );
		IF eState = eSOCKET_DISCONNECTED THEN
			sIpAdress:=fbConnect.sRemoteHost;
			fbReconnectTimer( IN := TRUE );(* Please wait some seconds and then try to connect again *)
			IF fbReconnectTimer.Q THEN
				fbReconnectTimer( IN := FALSE );
				nState := 0;
			END_IF
		END_IF

END_CASE

END_FUNCTION_BLOCK

// ---- POUs/Network Functions/UDP_Communication/FB_UDP_Server.TcPOU
FUNCTION_BLOCK FB_UDP_Server
VAR_IN_OUT
	IP_C : IP_C; (* IP_Control Verwaltungsstruktur *)
	S_BUF : ST_UDP_Buffer; (* Externer Sendbuffer *)
	R_BUF : ST_UDP_Buffer; (* Externer Receivebuffer *)
END_VAR
VAR_INPUT
	PORT 		: WORD; (* Port Nummer *)
	TIME_OUT 	: TIME; (* Ueberwachungszeit Connect / Send / Receive *)
	sLocal_IP	: T_IPv4Addr;
END_VAR
VAR_OUTPUT
END_VAR
VAR

	UDP_Reset : FB_UDP_Server_RESET;	

	s_time : UDINT; (* SEND-Time    (Zeit seit letzten Datensenden) *)
	r_time : UDINT; (* RECEIVE-Time (Zeit seit letztem Datenempfang) *)

	c_enable : BOOL; (* Connect: freigabe *)
	c_port : WORD; (* Connect: aktuelle Port-Nummer *)
	c_status : BYTE; (* Connect: Status (Errorcode) *)
	c_ready : BOOL; (* Connect: Verbindung aufgebaut *)
	c_ready_old : BOOL; (* Connect: letzter Zustand von c_ready für Flankenauswertung *)

	s_total : INT; (* Send: Gesamtanzahl Bytes zum senden *)
	s_cur_pos : INT; (* Send: aktuelle Sendeposition *)
	s_cur_size : INT; (* Send: aktuelle Sendegroesse *)
	s_max_size : INT; (* Send: maximale Telegrammlänge fuer Senden *)
	s_active : BOOL; (* Send: Daten senden ist aktiv *)
	s_status : BYTE; (* Send: Status (Errorcodes) *)
	r_status : BYTE; (* Receive: Status (Errorcodes) *)
	r_count : INT; (* Receive: Anzahl empfangener Bytes *)
	r_offset : INT; (* Receive: aktuelle Position in externen Receivebuffer *)
	r_max_size : INT; (* Receive: groesse des externen Empfangbuffers*)

	new_connection : BOOL; (* Neue Verbindungsparameter vorhanden *)
	tx : DWORD; (* letzter zeitwert *)
	error_time : DWORD; (* aktueller Timeout-Wert *)
	nErrId : UDINT;

	Send_Busy : BOOL;
	Send_Error : BOOL;
	Send_ErrId : UDINT;
	
	state: BYTE; (* schrittmerker für connect *)
	bytes_received : DINT;

	socket : T_HSOCKET;
	server : T_HSOCKET;
	fbCreate	: FB_SocketUdpCreate;	
	fbClose : FB_SocketClose;
	fbSendTo : FB_SocketUdpSendTo;
	fbReceiveFrom : FB_SocketUdpReceiveFrom;
	
END_VAR

VAR CONSTANT
	STOP : BYTE := 0;
	UDP_INIT : BYTE:= 31;
	UDP_INIT_WAIT : BYTE:= 32;
	C_CLOSE : BYTE := 190;
	C_CLOSE_WAIT : BYTE:= 191;
	C_CLOSE2 : BYTE := 192;
	C_CLOSE_WAIT2 : BYTE:= 193;
	C_WAIT : BYTE := 200;
	C_REC : BYTE := 210;
	C_REC_WAIT : BYTE := 211;
	C_SND : BYTE := 220;
	C_SND_WAIT1 : BYTE := 221;
	C_SND_WAIT2 : BYTE := 222;
END_VAR

(* Bei PLC reset oder Programm Download werden alle alten Verbindungen geschlossen *)
UDP_Reset();
IF NOT UDP_Reset.READY THEN RETURN; END_IF;

(* read system time *)
tx := TIME_TO_DWORD(TIME());

IF IP_C.C_PORT = 0 THEN
	IP_C.C_PORT := PORT; (* uebergebenen PORT durch parametrierten PORT ersetzen *)
END_IF;


new_connection := c_port <> IP_C.C_PORT; (* neue Verbindungs erwünscht ? *)
c_enable := IP_C.C_ENABLE AND NOT new_connection;

IF IP_C.C_ENABLE AND IP_C.ERROR = 0 AND state = STOP THEN (* Freigabe,kein Fehler,kein Socket offen *)
	c_port := IP_C.C_PORT;

	error_time := TIME_TO_DWORD(MAX(T#200ms,TIME_OUT));
	IP_C.TIME_RESET := TRUE; (* Alle Timer ruecksetzen *)
	r_max_size := UINT_TO_INT(SIZEOF(R_BUF.BUFFER));
	s_max_size := UINT_TO_INT(SIZEOF(S_BUF.BUFFER));

	(* Mode:  UDP CLIENT/SERVER *)
	state := UDP_INIT;


END_IF;

IF IP_C.TIME_RESET THEN (* Alle Timer ruecksetzen *)
	IP_C.TIME_RESET := FALSE; (* Reset rücksetzen *)
	s_time := tx; (* Send Timer ruecksetzen *)
	r_time := tx; (* Receive Timer ruecksetzen *)

	c_status := BYTE#0; (* letzten Connect Fehler rücksetzen *)
	s_status := BYTE#0; (* letzten Send Fehler rücksetzen *)
	r_status := BYTE#0; (* letzten Receive Fehler rücksetzen *)
END_IF;

(* ---------------------------------------------- *)

CASE state OF

UDP_INIT: (* UDP_CLIENT + SERVER *)
	(* 1. bei UDP-Client wird als lokalport 0 vorgegeben, damit das System automatisch einen freien lokalen Port sucht
	    2. bei UDP Server muss der gewüschte lokalport verwendet werden *)

	fbCreate(bExecute := FALSE);
	fbCreate(bExecute := TRUE , sSrvNetId := '', sLocalHost := sLocal_IP , nLocalPort := c_port , tTimeOut := TIME_OUT);
	fbCreate.bExecute := FALSE; (* vorbelegung *)
	state := UDP_INIT_WAIT;

UDP_INIT_WAIT:
	fbCreate();
	IF NOT fbCreate.bBusy THEN
		IF NOT fbCreate.bError THEN
			socket := fbCreate.hSocket;
			c_ready := TRUE; (* Connected *)
			state := C_WAIT;
		ELSE
			c_status := 1; (* FB_SocketUdpCreate failed *)
			nErrId := fbCreate.nErrId;
			state := C_CLOSE;
		END_IF;
	END_IF;

C_CLOSE:
	c_ready := FALSE;
	IF socket.handle > 0 THEN
		fbClose(bExecute := FALSE );
		fbClose(bExecute := TRUE, sSrvNetId := '',	hSocket := socket);
		fbClose.bExecute := FALSE;
		state := C_CLOSE_WAIT;
	ELSE
		state:= C_CLOSE2;
	END_IF;

C_CLOSE_WAIT:
	fbClose();
	IF NOT fbClose.bBusy THEN
		socket := TCPADS_NULL_HSOCKET; (* Socket rücksetzen *)
		nErrId:= SEL(fbClose.bError,0,fbClose.nErrId);
		state:= C_CLOSE2;
	END_IF;

C_CLOSE2:
	IF server.handle > 0 THEN
		fbClose(bExecute := FALSE );
		fbClose(bExecute := TRUE, sSrvNetId := '',	hSocket := server);
		fbClose.bExecute := FALSE;
		state := C_CLOSE_WAIT2;
	ELSE
		state:= STOP;
	END_IF;

C_CLOSE_WAIT2:
	fbClose();
	IF NOT fbClose.bBusy THEN
		server := TCPADS_NULL_HSOCKET; (* Socket rücksetzen *)
		nErrId:= SEL(fbClose.bError,0,fbClose.nErrId);
		state:= STOP;
	END_IF;

(* ---------------------------------------------- *)

C_WAIT: (* Warten auf Anforderung für Beenden *)
	IF NOT c_enable OR NOT c_ready THEN
		state:= C_CLOSE;
	ELSIF S_BUF.SIZE > 0 AND IP_C.MAILBOX[2] = 0 THEN
		state:= C_SND;
	ELSIF IP_C.MAILBOX[3] = 0 THEN
		state:= C_REC;
	END_IF;

(* ---------------------------------------------- *)

C_REC: (* Daten empfangen *)
	IF R_BUF.SIZE >= INT_TO_UINT(r_max_size) THEN
		R_BUF.SIZE := UINT#0;
		r_status := 254; (* Empfangsbuffer wegen Überlauf rückgesetzt *)
	END_IF;

	r_count := r_max_size;
	bytes_received := 0;

		fbReceiveFrom(bExecute := FALSE );
		fbReceiveFrom(bExecute:= TRUE, sSrvNetId := '', hSocket:= socket, cbLen := INT_TO_UINT(r_count), pDest:= ADR(R_BUF.BUFFER), tTimeout:= TIME_OUT);
		fbReceiveFrom.bExecute := FALSE; (* Vorbelegung *)

	state := C_REC_WAIT;

C_REC_WAIT:
		fbReceiveFrom(); (* UDP Mode *)
		IF NOT fbReceiveFrom.bBusy THEN
			IF NOT fbReceiveFrom.bError THEN
				IF fbReceiveFrom.nRecBytes > 0 THEN
					bytes_received := UDINT_TO_DINT(fbReceiveFrom.nRecBytes);
					R_BUF.Ip_Adresss 		:= fbReceiveFrom.sRemoteHost;
					R_BUF.nDriveMemberNr	:= WORD_TO_INT(WORD_OF_BYTE(B1:=R_BUF.BUFFER[0],B0:=R_BUF.BUFFER[1]));
					R_BUF.nPLCMemberNr		:= WORD_TO_INT(WORD_OF_BYTE(B1:=R_BUF.BUFFER[2],B0:=R_BUF.BUFFER[3]));
					R_BUF.SIZE 				:= UDINT_TO_UINT(fbReceiveFrom.nRecBytes); (* aktuelle buffersize eintragen *)
				END_IF;
				state := C_WAIT;
			ELSIF fbReceiveFrom.nErrId = 16#80072746 THEN (* Verbindung vom Remote beendet *)
				c_status := 253;
				c_ready := FALSE;
				state := C_WAIT;
			ELSE
				nErrId := fbReceiveFrom.nErrId;
				state := C_WAIT;
			END_IF;
		END_IF;

	IF bytes_received > 0 THEN
		r_time := tx; (* Receive Timer ruecksetzen *)
		IP_C.MAILBOX[1] := IP_C.MAILBOX[1] + 1; (* Receive Info *)
		IF IP_C.MAILBOX[1] = 0 THEN IP_C.MAILBOX[1] := 1; END_IF;
	END_IF;

(* ---------------------------------------------- *)
C_SND:
	IF S_BUF.SIZE > 0 THEN
		IF c_ready AND c_enable THEN
			IF NOT s_active THEN
				s_total := LIMIT(0,UINT_TO_INT(S_BUF.SIZE),r_max_size); (* Gesamtanzahl an Bytes limitieren und uebergeben *)
				s_cur_pos  := 0;
				s_cur_size := 0;
				s_active := TRUE; (* Sende-Betrieb aktivieren *)
			END_IF;

			s_cur_pos := s_cur_pos + s_cur_size; (* neue Sende-Datenposition bestimmen *)
			IF s_total > s_cur_pos THEN (* weitere Daten zum senden vorhanden ? *)
				s_cur_size := s_total - s_cur_pos;
				s_cur_size := LIMIT(0, s_cur_size, s_max_size); (* Telegrammlänge begrenzen *)
				s_time := tx; (* Send Timer ruecksetzen *)
				r_time := tx; (* Receive Timer ruecksetzen *)
				state := C_SND_WAIT1;
			ELSE (* keine weitere Sendedaten vorhanden -> Senden beenden *)
				s_active := FALSE;
				S_BUF.SIZE := 0;
				state := C_WAIT;
			END_IF;
		END_IF;
	END_IF;

C_SND_WAIT1:
		fbSendTo(bExecute := FALSE );
		fbSendTo(bExecute := TRUE, sSrvNetId := '', hSocket := socket , cbLen := INT_TO_UDINT(s_cur_size), pSrc := ADR(S_BUF.BUFFER[s_cur_pos]), sRemoteHost := S_BUF.Ip_Adresss, nRemotePort := c_port, tTimeout:= TIME_OUT);
		fbSendTo.bExecute := FALSE;
	state := C_SND_WAIT2;

C_SND_WAIT2:

		fbSendTo();
		Send_Busy := fbSendTo.bBusy;
		Send_Error := fbSendTo.bError;
		Send_ErrId := fbSendTo.nErrId;


	IF NOT Send_Busy THEN
		IF NOT Send_Error THEN
			state := C_SND;
		ELSE
			nErrId := Send_ErrId;
			state := C_WAIT;
		END_IF;
	END_IF;

END_CASE;

(* ---------------------------------------------- *)

IF c_ready THEN
	IF NOT c_ready_old THEN (* Verbindung aufgebaut - positive Flanke erkannt *)
		IP_C.C_STATE := 254;
		IP_C.TIME_RESET := TRUE; (* Alle Timer ruecksetzen *)
	ELSE
		IP_C.C_STATE := 255; (* Verbindung ist aufgebaut *)
	END_IF;
ELSE
	IF c_ready_old THEN (* Verbindung abgebaut - negative Flanke erkannt *)
		IP_C.C_STATE := 1;
		IP_C.MAILBOX[1] := 0; (* Receive Info rücksetzen *)
		IP_C.MAILBOX[2] := 0; (* Send-Pause rücksetzen *)
		IP_C.MAILBOX[3] := 0; (* Receive-Pause rücksetzen *)
		IF NOT new_connection THEN
			s_active := FALSE; (* Sendeaktivitäten stoppen *)
			S_BUF.SIZE := 0; (* Sendelänge löschen *)
			(*IP_C.TIME_RESET := TRUE; *) (* Alle Timer ruecksetzen *)
		END_IF;

	ELSE
		IP_C.C_STATE := 0; (* Verbindung ist abgebaut *)
	END_IF;
END_IF;

c_ready_old := c_ready;

(* ---------------------------------------------- *)

IF IP_C.R_OBSERVE = FALSE OR s_active THEN
    r_time := tx;
END_IF;

IF s_status = 0 AND tx - s_time > error_time AND s_active THEN (* Send Timeout *)
	s_status := 255; (* Timeout-Fehler ausgeben *)
END_IF;
IF r_status = 0 AND tx - r_time > error_time AND c_ready AND IP_C.R_OBSERVE THEN (* Receive Timeout *)
	r_status := 255; (* Timeout-Fehler ausgeben *)
END_IF;

IP_C.ERROR := DWORD_OF_BYTE(c_status,s_status,r_status,0);

END_FUNCTION_BLOCK

// ---- POUs/Network Functions/UDP_Communication/FB_UDP_Server_RESET.TcPOU
FUNCTION_BLOCK FB_UDP_Server_RESET
VAR_INPUT
END_VAR
VAR_OUTPUT
	READY : BOOL;
END_VAR
VAR
	fbSocketCloseAll : FB_SocketCloseAll;
	step : BYTE;
END_VAR

(* On PLC reset or program download close all old connections *)

CASE UDP_SERVER_RESET OF

2:	READY := TRUE;
	RETURN;

1:	IF step = 0 THEN
		RETURN;
	END_IF;

0:	UDP_SERVER_RESET := 1; (* Reset ist aktiv *)
	step := 1;

END_CASE;

CASE step OF

0:	RETURN;

1:	fbSocketCloseAll(sSrvNetId:= '', bExecute:= TRUE, tTimeout:= T#10s );
	step := 2;

2:	fbSocketCloseAll(bExecute:= FALSE);
	IF fbSocketCloseAll.bBusy = FALSE THEN
		step := 0;
		UDP_SERVER_RESET := 2; (* Reset durchgeführt , Bereit zur Verwendung *)
	END_IF;

END_CASE;

END_FUNCTION_BLOCK

// ---- POUs/UDFB/DWORD_OF_BYTE.TcPOU
FUNCTION DWORD_OF_BYTE : DWORD
VAR_INPUT
	B3 : BYTE;
	B2 : BYTE;
	B1 : BYTE;
	B0 : BYTE;
END_VAR


(*
version 1.3	18. jul. 2009
programmer 	hugo
tested by		tobias

this function creates a Dword from 4 individual bytes

*)

DWORD_OF_BYTE := SHL(SHL(SHL(BYTE_TO_DWORD(B3),8) OR BYTE_TO_DWORD(B2),8) OR BYTE_TO_DWORD(B1),8) OR BYTE_TO_DWORD(B0);


(* revision history
hm	24. jan 2007	rev 1.0
	original version

hm 2. jan 2008	rev 1.1
	inproved performance

hm	23. apr. 2008	rev 1.2
	reverse order of inputs to be more logical

hm	18. jul. 2009	rev 1.3
	added type conversions for compatibility reasons
*)

END_FUNCTION

// ---- POUs/Pecom Interface/PB_Start_TCPIP.TcPOU
PROGRAM PB_Start_TCPIP
VAR_INPUT	
	sLocal_IP		: T_Ipv4Addr;	// IP-Adress of the the local Ethernetport where we want to listen/Send
	Setup_MdsCom	: POINTER TO  ARRAY [0..20] OF ST_SetupDriveComMDS;
END_VAR
VAR_IN_OUT
	iResetTCP		: BOOL;	
END_VAR
VAR
	
(****************************************************************)
(*******		TCP Passiv Listener Functions				*****)	
(****************************************************************)

	sSrvNetID		: T_AmsNetID	:= '';(* TwinCAT TCP/IP server network address *)
	nLocalPort		: UDINT 		:= 8101;(* Server port number *)
	bLog			: BOOL			:= FALSE;(* TRUE => Enable log message output, FALSE => Disable *)
	afbServer		: ARRAY[1..NR_OF_DRIVEMASTERS] OF FB_Server;(* Server (connection) instance *)
	hServer			: T_HSERVER;(* Server connection handle *)

(****************************************************************)	
	
	fbCloseAll	: FB_SocketCloseAll;
	bInitialize	: BOOL := TRUE;
	
	(* Pecom Communication for desk A and B *)
	FB_SendReceive_TCP	:	ARRAY[1..NR_OF_DRIVEMASTERS] OF FB_SendReceive_TcpIp;
	
	IP_Adr_A: DWORD;


	nCount: INT;
	nBuffer				: ARRAY[0..NR_OF_DRIVEMASTERS] OF INT;
	nBuffer_empty		: ARRAY[0..NR_OF_DRIVEMASTERS] OF INT;
	n: INT;
	sServerPrefix: STRING;
	nIP_SetupCount: INT;
	bServerHandleState: BOOL;
	TON_ResetConnection: TON;
END_VAR

(* On PLC reset or program download close all old (opened) connections *)
TON_ResetConnection(IN:=iResetTCP, PT:=T#3S);
IF iResetTCP AND TON_ResetConnection.Q THEN
	bInitialize	:= TRUE;
	iResetTCP	:= FALSE;
END_IF
fbCloseAll( sSrvNetID := sSrvNetID, bExecute:= iResetTCP );
IF fbCloseAll.bBusy OR fbCloseAll.bError THEN
	RETURN;
END_IF


IF bInitialize THEN
	bInitialize := FALSE;

	(* Initialize server handle *)
	bServerHandleState := F_CreateServerHnd( 	sSrvNetID 	:= sSrvNetID,
												sLocalHost 	:= sLocal_IP,
												nLocalPort	:= nLocalPort,
												nMode 		:= SEL( bLog, 0, CONNECT_MODE_ENABLEDBG ),(* Enable debug messages *)
												bEnable 	:= TRUE,(* TRUE = leave listener socket open, FALSE = close listener socket after last connection ist closed too *)
												hServer 	:= hServer );	
END_IF




(* Trigger the execution of every server (connection) instance *)
FOR n := 1 TO NR_OF_DRIVEMASTERS DO
	sServerPrefix := Concat('SERVER',INT_TO_STRING(n));
	sServerPrefix := Concat(sServerPrefix,':: ');
	afbServer[n] ( hServer := hServer, sSrvNetID := sSrvNetID, bEnable := TRUE, bLog := bLog, nServer_Id := n, sPrefix := sServerPrefix );
	stComStatus.bTCP_Connect[n] := FALSE;
END_FOR

nBuffer := nBuffer_empty;
FOR nCount:= 1 TO NR_OF_DRIVEMASTERS DO
	FOR nIP_SetupCount:= 1 TO NR_OF_DRIVEMASTERS DO
		IF aTcpPuff[nCount].Ip_Adresss = Setup_MdsCom^[nIP_SetupCount].stSetup_MDS_IP 
			AND aTcpPuff[nCount].Ip_Adresss <> ''
			THEN
				nBuffer[nIP_SetupCount] 			:= nCount;
				aTcpPuff[nCount].PecomTNR 			:= Setup_MdsCom^[nIP_SetupCount].nPLCMemberNr_1;
				stComStatus.bTCP_Connect[nCount]	:= TRUE;	// Write Status
		END_IF
	END_FOR	
END_FOR
(**********************************************)
(***			Diagnose only				***)
(**********************************************)
Setup_MdsCom^[1].stSetup_MDS_IP;
Setup_MdsCom^[2].stSetup_MDS_IP;
Setup_MdsCom^[3].stSetup_MDS_IP;
Setup_MdsCom^[4].stSetup_MDS_IP;
Setup_MdsCom^[5].stSetup_MDS_IP;
Setup_MdsCom^[6].stSetup_MDS_IP;
Setup_MdsCom^[7].stSetup_MDS_IP;
Setup_MdsCom^[8].stSetup_MDS_IP;
Setup_MdsCom^[9].stSetup_MDS_IP;
Setup_MdsCom^[10].stSetup_MDS_IP;
Setup_MdsCom^[1].nPLCMemberNr_1;
Setup_MdsCom^[2].nPLCMemberNr_1;
Setup_MdsCom^[3].nPLCMemberNr_1;
Setup_MdsCom^[4].nPLCMemberNr_1;
Setup_MdsCom^[5].nPLCMemberNr_1;
Setup_MdsCom^[6].nPLCMemberNr_1;
Setup_MdsCom^[7].nPLCMemberNr_1;
Setup_MdsCom^[8].nPLCMemberNr_1;
Setup_MdsCom^[9].nPLCMemberNr_1;
Setup_MdsCom^[10].nPLCMemberNr_1;

(**********************************************)
(***			Diagnose only				***)
(**********************************************)
aTcpPuff[nBuffer[1]].Ip_Adresss;
aTcpPuff[nBuffer[1]].PecomTNR;
aTcpPuff[nBuffer[1]].Conected;
aTcpPuff[nBuffer[1]].R_Buf.SIZE; 

aTcpPuff[nBuffer[2]].Ip_Adresss;
aTcpPuff[nBuffer[2]].PecomTNR;
aTcpPuff[nBuffer[2]].Conected;
aTcpPuff[nBuffer[2]].R_Buf.SIZE;
               
aTcpPuff[nBuffer[3]].Ip_Adresss;
aTcpPuff[nBuffer[3]].PecomTNR;
aTcpPuff[nBuffer[3]].Conected;
aTcpPuff[nBuffer[3]].R_Buf.SIZE;
               
aTcpPuff[nBuffer[4]].Ip_Adresss;
aTcpPuff[nBuffer[4]].PecomTNR;
aTcpPuff[nBuffer[4]].Conected;
aTcpPuff[nBuffer[4]].R_Buf.SIZE;
              
aTcpPuff[nBuffer[5]].Ip_Adresss;
aTcpPuff[nBuffer[5]].PecomTNR;
aTcpPuff[nBuffer[5]].Conected;
aTcpPuff[nBuffer[5]].R_Buf.SIZE;

aTcpPuff[nBuffer[6]].Ip_Adresss;
aTcpPuff[nBuffer[6]].PecomTNR;
aTcpPuff[nBuffer[6]].Conected;
aTcpPuff[nBuffer[6]].R_Buf.SIZE;

aTcpPuff[nBuffer[7]].Ip_Adresss;
aTcpPuff[nBuffer[7]].PecomTNR;
aTcpPuff[nBuffer[7]].Conected;
aTcpPuff[nBuffer[7]].R_Buf.SIZE;

aTcpPuff[nBuffer[8]].Ip_Adresss;
aTcpPuff[nBuffer[8]].PecomTNR;
aTcpPuff[nBuffer[8]].Conected;
aTcpPuff[nBuffer[8]].R_Buf.SIZE;

aTcpPuff[nBuffer[9]].Ip_Adresss;
aTcpPuff[nBuffer[9]].PecomTNR;
aTcpPuff[nBuffer[9]].Conected;
aTcpPuff[nBuffer[9]].R_Buf.SIZE;

aTcpPuff[nBuffer[10]].Ip_Adresss;
aTcpPuff[nBuffer[10]].PecomTNR;
aTcpPuff[nBuffer[10]].Conected;
aTcpPuff[nBuffer[10]].R_Buf.SIZE;

(************************************************)
(***** TCP communication remote System 1..x	*****)
FOR n := 1 TO NR_OF_DRIVEMASTERS DO
	IF Setup_MdsCom^[n].nPLCMemberNr_1 > 0 THEN 
		FB_SendReceive_TCP[n]( R_BUF_A 				:= aTcpPuff[nBuffer[n]].R_Buf,
							   S_BUF_A				:= aTcpPuff[nBuffer[n]].S_Buf,
							   iConnected 			:= aTcpPuff[nBuffer[n]].Conected,
							   nPecom_Tnr_Remote_1	:= Setup_MdsCom^[n].nPLCMemberNr_1,
							   nPecom_Tnr_Remote_2	:= Setup_MdsCom^[n].nPLCMemberNr_2,
							   nPecom_Tnr_Local		:= Setup_MdsCom^[n].nDriveMemberNr);
	END_IF
END_FOR

(***************************************************************)
(*******  This starts the Pecom Protokoll Functions		********)
Eth_Send_Receive();
Pecom_In_Out_data();	// Pecom Communication Layer

END_PROGRAM

// ---- POUs/Pecom Interface/Pecom_Functions/TCP Msg Handling/FB_SendReceive_TcpIp.TcPOU
FUNCTION_BLOCK   FB_SendReceive_TcpIp
VAR_INPUT	
    iConnected	: BOOL;
	nPecom_Tnr_Remote_1	: INT;		// pecom member number of the remote partner (LST or PLC)
	nPecom_Tnr_Remote_2	: INT;		// pecom member number of the remote partner (LST or PLC)
	nPecom_Tnr_Local	: INT;		// Own pecom member number for the member anouncement (Teilnehmerauskunft)
END_VAR
VAR_IN_OUT	
	S_BUF_A				:	NETWORK_BUFFER;
	R_BUF_A				:	NETWORK_BUFFER;
END_VAR

VAR
	IP_TNA				:	ST_MemberAnounce;
	Rec_Buffer			:	ARRAY [0..1400] OF WORD;
	R_TRIG_Connected	:	R_TRIG;
	k					:	INT;
	N					:	INT;
	i					:	INT;
	M					:	INT;
	message_in			:	BOOL;
	buffer_length		:	INT;
	nPointer			:	INT;
	msg_count			:	INT;
	nMSG_Length			:	INT;
	IN_pointer			:	INT;
	counter				:	INT;
	nCountMessage		:	INT;	
	state				:	INT;
	start_init			:	BOOL;
END_VAR

(************************************************************************************************************)
(*********** 		Ethernet Communication 														*************)
(************************************************************************************************************)

(* Ethernetverbindung aufbauen *)
(* This is for connecting over the Ethernet. The first desk is called "A". Normally this is the Pecom number 71. *)
(* The Oscat library works with the IP_C and with IP_Control *)
(* For sending a message we have to fill the buffer and after that write into S_BUF_A.SIZE the length *)
(* this is the command for sending the buffer *)
(* to look for an incoming message we have to lokk into R_BUF_A.SIZE and if it is not zero we have a new message *)
(* The Byte must be switched to get them into a Word *)

(*************************************)
(* Connection *)
R_TRIG_Connected(CLK:=	iConnected);
start_init :=	R_TRIG_Connected.Q;


(************************************************************************************************************)
(*********** 		Ethernetkommunikation 														*************)
(************************************************************************************************************)
(* This is on a low level of the Pecom communication *)
(* after starting a new connection we have to tell the remote partner what Pecom number we have and the partner *)  
(* system takes this number into his own member list *)
(* with this message the remote partner system can do the relationsship from the IP adress to the member number *)
(* sender and receiver is always 65535, only for this message the type is 7, normally this is 153 *)

(******************************************************)
(* Pecom Member Announcement/ build the message 65535 *)
(******************************************************)
CASE	state OF
	00:
		IF start_init THEN
			state := state + 2;	
		END_IF
	02:
	
		IP_TNA.Laenge := WORD#12;
		IP_TNA.receiver := WORD#65535;
		IP_TNA.Sender := WORD#65535;
		IP_TNA.Typ := WORD#7; (*must be 7 not 153 *)
		IP_TNA.Reserve := WORD#0;
		IP_TNA.N_Laenge := WORD#02;
		IP_TNA.Kommando := INT_TO_WORD(nPecom_Tnr_Local);
		state := 10;
	
	10:
		R_BUF_A.SIZE	:=	UINT#0;	// Reset the Receiver Buffer, so rest will not be read
	
	
		S_BUF_A.BUFFER[0] := WORD_TO_BYTE(SHR(IP_TNA.receiver,8));
		S_BUF_A.BUFFER[1] := WORD_TO_BYTE(IP_TNA.receiver);
		S_BUF_A.BUFFER[2] := WORD_TO_BYTE(SHR(IP_TNA.Sender,8));
		S_BUF_A.BUFFER[3] := WORD_TO_BYTE(IP_TNA.Sender);
	
		S_BUF_A.BUFFER[4] := WORD_TO_BYTE(SHR(IP_TNA.Typ,8));
		S_BUF_A.BUFFER[5] := WORD_TO_BYTE(IP_TNA.Typ);
	
		S_BUF_A.BUFFER[6] := WORD_TO_BYTE(SHR(IP_TNA.Reserve,8));
		S_BUF_A.BUFFER[7] := WORD_TO_BYTE(IP_TNA.Reserve);
	
		S_BUF_A.BUFFER[8] := WORD_TO_BYTE(SHR(IP_TNA.N_Laenge,8));
		S_BUF_A.BUFFER[9] := WORD_TO_BYTE(IP_TNA.N_Laenge);
	
		S_BUF_A.BUFFER[10] := WORD_TO_BYTE(SHR(IP_TNA.Kommando,8));
		S_BUF_A.BUFFER[11] := WORD_TO_BYTE(IP_TNA.Kommando);
	
	
		S_BUF_A.SIZE := (IP_TNA.Laenge);
	state	:=	30;
	
	30:
		state	:=	0;

END_CASE;


(************************************************************************************************************)
(********** Send                                           											*********)
(************************************************************************************************************)
(* TCP *)

k	:=	0;
IF	S_BUF_A.SIZE	=	UINT#0
THEN
	FOR	N := 1 TO	40
	DO
		IF	st_OUT_PecomMsg.valid[N]
			AND	(st_OUT_PecomMsg.stMsgBuffer[N].MSG[0]	=	INT_TO_WORD(nPecom_Tnr_Remote_1)
				OR st_OUT_PecomMsg.stMsgBuffer[N].MSG[0]	=	INT_TO_WORD(nPecom_Tnr_Remote_2))
		THEN
			st_OUT_PecomMsg.stMsgBuffer[N].MSG[1]	:= INT_TO_WORD(nPecom_Tnr_Local);
			FOR	i	:= 0 TO (WORD_TO_INT(st_OUT_PecomMsg.stMsgBuffer[N].MSG[4]) / 2) + 4
			DO
				S_BUF_A.BUFFER[k]		:=	WORD_TO_BYTE(SHR(st_OUT_PecomMsg.stMsgBuffer[N].MSG[i],8));
				k	:=	k + 1;
				S_BUF_A.BUFFER[k]		:=	WORD_TO_BYTE(st_OUT_PecomMsg.stMsgBuffer[N].MSG[i]);
				k	:=	k + 1;
			END_FOR;
			st_OUT_PecomMsg.number_of_buffers	:=	st_OUT_PecomMsg.number_of_buffers + 1;
			st_OUT_PecomMsg.valid[N]	:=	FALSE;
		END_IF;
	END_FOR;
		S_BUF_A.SIZE	:=	INT_TO_UINT(k);			(* send with write  into the size-Byte*)
END_IF;

(************************************************************************************************************)
(********** Receive Messages																		*********)
(************************************************************************************************************)
(* TCP *)
IF		R_BUF_A.SIZE >= UINT#1
THEN	(* Clear and Read Receiver-Buffer first *)
	FOR i := 0 TO 700 DO	// Clear
		Rec_Buffer[i] := WORD#0;
	END_FOR;
	k	:= 0;
	FOR i := 0 TO	UINT_TO_INT(R_BUF_A.SIZE)/2 DO // Read
		Rec_Buffer[i]	:=	WORD_OF_BYTE(R_BUF_A.BUFFER[k],R_BUF_A.BUFFER[k+1]);
		k	:= k + 2;
	END_FOR;
	message_in	:=	TRUE;
	buffer_length	:=	UINT_TO_INT(R_BUF_A.SIZE)/2;
	R_BUF_A.SIZE		:=	UINT#0;
	counter	:=	counter + 1;		// Diagnose counter for incoming trafic

END_IF;


(************************************************************************************************************)
(********** Sort incomming messages into the In-Buffer												*********)
(************************************************************************************************************)
(* Sort incomming messages into the In-Buffer                                   *)
(* max. 40 incoming messages can be sorted in 1 cycle					        *)
(* from IN_MSG1.MESS[1..40].MSG[0..49] 					                        *)
(* In IN_MSG1.valid[1..40] steht für 1 Zyklus die validkeit                 	*)
(********************************************************************************)

(* in one message (in one buffer) can be a lot of normal Pecom messages *)
(* so we have to look for them and sort them into extra buffers to work with them *)
(* we have 40 extra buffers and if we have put a new Pecom message into one we have to set the Bit IN_MSG1.valid[M] *)
(* this also usefull if the cycletime of the PLC is to slow. We never can loose a message if the numbers of the buffers are big anough *)

IF message_in = TRUE THEN    
	
		nPointer := 0;
		msg_count := 0;
		
		FOR M := 1 TO 40
		DO
			IF NOT st_IN_PecomMsg.valid[M]
			THEN
				IF buffer_length >= 6
				THEN
					nMSG_Length := msg_count + 4;
					FOR IN_pointer := (0 + msg_count) TO (WORD_TO_INT(Rec_Buffer[nMSG_Length]) / 2) + 4 + msg_count
					DO
						nPointer := IN_pointer - msg_count;
						st_IN_PecomMsg.stMsgBuffer[M].MSG[nPointer] := Rec_Buffer[IN_pointer];
						buffer_length := buffer_length - 1;
					END_FOR;
					msg_count := IN_pointer;
					st_IN_PecomMsg.valid[M] := TRUE;
					nCountMessage := nCountMessage + 1;
				END_IF;
			END_IF;
		END_FOR;
		
		IF buffer_length > 0
		THEN
			st_IN_PecomMsg.buffer_overfow := TRUE;
		END_IF;
	
		st_IN_PecomMsg.number_of_buffers	:=	nCountMessage;
		message_in := FALSE;
END_IF;

END_FUNCTION_BLOCK

// ---- POUs/Pecom Interface/Pecom_Functions/TCP Msg Handling/Eth_Send_Receive.TcPOU
PROGRAM Eth_Send_Receive
VAR
	Ethernet_Receive_Objects:	FB_Msg_Receive;
	Ethernet_Send_Objects:	FB_Msg_Send;

	OBJ_receiver:	INT;
	OBJ_Nachricht:	BOOL;
	OBJ_Nachricht_senden:	BOOL;
	OBJ_Nachricht_an_LST_A:	BOOL;

	Test:	BOOL;

	MSG_receiver: INT;
	Ethernet_Send_LST_SH: FB_Msg_Send;
END_VAR
VAR_OUTPUT
	SH_Nachricht_an_LST_A: BOOL;
END_VAR

TCP_PecomOBJ();
TCP_Alarms();

ACTION TCP_Alarms:
(*-- Send MSG --*)
IF	MSG_receiver = 0
	AND NOT st_OUT_Alarms_Buffer.data_transfer_ready
	AND st_OUT_Alarms_Buffer.data_are_valid	
	THEN	
		MSG_receiver 			:= 	st_OUT_Alarms_Buffer.receiver;
END_IF;

IF		MSG_receiver = 0
	THEN	
		IF	st_OUT_Alarms_Buffer.data_are_valid
			THEN
				st_OUT_Alarms_Buffer.receiver 			:= 	INT#0;
				st_OUT_Alarms_Buffer.data_are_valid 	:= 	FALSE;
		END_IF;
END_IF;

Ethernet_Send_LST_SH ( 	receiver 	:= 	MSG_receiver,
				       	Sender	  	:= 	st_OUT_Alarms_Buffer.Sender,
				       	Freigabe	:= 	st_OUT_Alarms_Buffer.data_are_valid,
				       	Typ		  	:= 	'TCP',
				       	Puffer	  	:= 	st_OUT_Alarms_Buffer);
st_OUT_Alarms_Buffer.nNumber_of_messages; 	(*Diagnose*)
st_OUT_Alarms_Buffer.nNumber_of_Error; 		(*Diagnose*)


IF	(	st_OUT_Alarms_Buffer.job_done
	OR	st_OUT_Alarms_Buffer.job_not_done )
	AND	st_OUT_Alarms_Buffer.data_transfer_ready
	THEN	(* message done *)
		MSG_receiver 							:= 0;
		st_OUT_Alarms_Buffer.data_transfer_ready 	:= FALSE;
		st_OUT_Alarms_Buffer.receiver 				:= INT#0;
		st_OUT_Alarms_Buffer.data_are_valid 		:= FALSE;
END_IF;
END_ACTION

ACTION TCP_PecomOBJ:
(*--- Receive  ---*)
Ethernet_Receive_Objects(	Freigabe	:= TRUE,
							Typ			:= 'TCP',
							Puffer		:= st_IN_Objects);

st_IN_Objects.nNumber_of_messages := st_IN_Objects.nNumber_of_messages; (*Diagnose*)


(*--------------------------------------------------------------------------------------------------*)
(*-- Send  --*)
IF		st_OUT_Objects_Buffer.receiver >	0
	AND	OBJ_receiver = 0
	AND	NOT	OBJ_Nachricht_senden
	AND st_OUT_Objects_Buffer.data_are_valid	
	THEN
		OBJ_Nachricht	:= TRUE;
		OBJ_receiver	:= st_OUT_Objects_Buffer.receiver;
END_IF;

(*-- 1 cycle later --*)
OBJ_Nachricht_senden	:=	OBJ_receiver <> 0;

Ethernet_Send_Objects(	receiver 	:= 	OBJ_receiver,
				       	Sender	  	:= 	0,
				       	Freigabe	:= 	OBJ_Nachricht_senden,
				       	Typ		  	:= 	'TCP',
				       	Puffer	  	:= 	st_OUT_Objects_Buffer);
st_OUT_Objects_Buffer.nNumber_of_messages; 	(*Diagnose*)
st_OUT_Objects_Buffer.nNumber_of_Error; 	(*Diagnose*)

IF	(	st_OUT_Objects_Buffer.job_done
	OR	st_OUT_Objects_Buffer.job_not_done)
	AND st_OUT_Objects_Buffer.data_transfer_ready
	THEN	
		OBJ_receiver 									:= 	0;
		st_OUT_Objects_Buffer.data_transfer_ready 		:=	FALSE;

		IF 		OBJ_Nachricht
			THEN
				st_OUT_Objects_Buffer.data_are_valid	:=	FALSE;
				st_OUT_Objects_Buffer.receiver			:=	INT#0;
				OBJ_Nachricht 							:=	FALSE;
		END_IF;
END_IF;
END_ACTION

END_PROGRAM

// ---- POUs/Pecom Interface/Pecom_Functions/TCP Msg Handling/FB_Msg_Receive.TcPOU
FUNCTION_BLOCK FB_Msg_Receive
VAR_INPUT
	Freigabe			:	BOOL;
	Typ					:	STRING;
END_VAR
VAR_IN_OUT
	Puffer				:	ST_InOut_Data;
END_VAR
VAR
	Event_Error			:	INT;
	Nachrichtenlaenge	:	INT;
	TNR_neu				:	INT;
	N					:	INT;
	k					:	INT;
	i					:	INT;
END_VAR

(****** TCP ******************************************************************)
IF Typ = 'TCP' THEN
	
	IF NOT	Puffer.data_transfer_ready (* read data still running *)
	THEN	(* data read *)
		(*	
		IF 	Sender = 0 
			THEN
				RETURN; 
		END_IF;

		Puffer.receiver := receiver;
		IF		receiver <> -1 	THEN  (* Broadcast *)			
			Puffer.Sender := Sender; 
		END_IF;
		*)

		(********************************************************************************)
		(* Seek in IN_MSG for valif Msg and sort it into the Buffer                   	*)
		(********************************************************************************)
		(* Es koennen max. 40 Nachrichten gleichzeitig einsortiert werden und aus       *)
		(* IN_MSG1.MESS[1..40].MSG[0..99] ausgelesen werden.                            *)
		(* In IN_MSG1.valid[1..40] steht für 1 Zyklus die validkeit                 *)
		(********************************************************************************)

		(* Aus dem TCP Buffer die erste gültige Nachricht einlesen *)
		FOR	N:= 1	TO 40 DO
		  IF	st_IN_PecomMsg.valid[N]
		  THEN
			  IF NOT	Puffer.data_transfer_ready (* was read *)
			  THEN	(* data copy *)
				Puffer.receiver   := WORD_TO_INT(st_IN_PecomMsg.stMsgBuffer[N].MSG[0]);
				Puffer.Sender 	  := WORD_TO_INT(st_IN_PecomMsg.stMsgBuffer[N].MSG[1]);
				Puffer.Typ		  := WORD_TO_INT(st_IN_PecomMsg.stMsgBuffer[N].MSG[2]);
				Puffer.NFB		  := WORD_TO_INT(st_IN_PecomMsg.stMsgBuffer[N].MSG[3]);
				Puffer.Lg_Byte	  := WORD_TO_INT(st_IN_PecomMsg.stMsgBuffer[N].MSG[4]);
				Puffer.KDO		  := WORD_TO_INT(st_IN_PecomMsg.stMsgBuffer[N].MSG[5]);
				Nachrichtenlaenge := Puffer.Lg_Byte / 2 + 5;
				FOR i := 6 TO Nachrichtenlaenge
				DO 	k	:=	i + 1;
					Puffer.data[k] := WORD_TO_INT(st_IN_PecomMsg.stMsgBuffer[N].MSG[i]);
				END_FOR;
				st_IN_PecomMsg.valid[N]:= FALSE;
				Puffer.data_transfer_ready := TRUE;
				EXIT;
			 END_IF;
		  END_IF;
		END_FOR;
		
		FOR	N:= 1	TO 20 DO
		  IF	st_IN_PecomMsg.valid[N]
		  THEN
			IF	( WORD_TO_INT(st_IN_PecomMsg.stMsgBuffer[1].MSG[0]) = -1 )
					 AND ( WORD_TO_INT(st_IN_PecomMsg.stMsgBuffer[1].MSG[1]) = -1 )
				THEN
				TNR_neu	:=	 WORD_TO_INT(st_IN_PecomMsg.stMsgBuffer[1].MSG[5]);
				st_IN_PecomMsg.valid[1]:= FALSE;
				stComStatus.stRestart.TLN[1]	:=	TNR_neu;
				Puffer.data_transfer_ready := TRUE;
				EXIT;
			 END_IF;
			END_IF;
		END_FOR;
		
	END_IF; (* transfer_ready *)
	
END_IF; (* of TCP *)

END_FUNCTION_BLOCK

// ---- POUs/Pecom Interface/Pecom_Functions/TCP Msg Handling/FB_Msg_Send.TcPOU
FUNCTION_BLOCK FB_Msg_Send
VAR_INPUT
	receiver		:	INT;
	Sender			:	INT;
	Freigabe		:	BOOL;
	Typ				:	STRING;
END_VAR
VAR_OUTPUT
END_VAR
VAR_IN_OUT
	Puffer:	ST_InOut_Data;
END_VAR
VAR
	Puffer_receiver:	INT;
	Nachrichtenlaenge:	INT;
	N:	INT;
	i:	INT;
	k:	INT;
END_VAR

(****** TCP ******************************************************************)
IF Typ = 'TCP'
THEN	
	IF 	NOT Puffer.data_transfer_ready
		AND Freigabe
	THEN	
		Puffer.job_running 			:= TRUE;
		Puffer.job_done 			:= FALSE;
		Puffer.job_not_done 		:= FALSE;
		Puffer.data_transfer_ready 	:= TRUE;
		Puffer.nNumber_of_messages 	:= Puffer.nNumber_of_messages + 1; (* Diagnosezaehler *)
		
		Puffer_receiver				:=	Puffer.receiver;
		Puffer.receiver				:= 	receiver;
		Puffer.Sender				:= 	Sender;
	
		(* to send a message to the desk we also have an array of buffers *)
		(* we can use 40 buffers *)
		(* In OUT_MSG1.MESS[N].MSG[0] we have the desk number, so we can sort out were to we have to send them *)
		FOR	N	:=	1	TO	40 DO
			IF	st_OUT_PecomMsg.valid[N]	=	FALSE
			THEN
				st_OUT_PecomMsg.stMsgBuffer[N].MSG[0] := INT_TO_WORD(Puffer.receiver);
				st_OUT_PecomMsg.stMsgBuffer[N].MSG[1] := INT_TO_WORD(Puffer.Sender) ;
				st_OUT_PecomMsg.stMsgBuffer[N].MSG[2] := INT_TO_WORD(Puffer.Typ) ;
				st_OUT_PecomMsg.stMsgBuffer[N].MSG[3] := INT_TO_WORD(Puffer.NFB) ;
				st_OUT_PecomMsg.stMsgBuffer[N].MSG[4] := INT_TO_WORD(Puffer.Lg_Byte) ;
				st_OUT_PecomMsg.stMsgBuffer[N].MSG[5] := INT_TO_WORD(Puffer.KDO) ;
				Nachrichtenlaenge := Puffer.Lg_Byte / 2 + 5; 
				FOR	i := 6 TO Nachrichtenlaenge DO	
					k	:=	i + 1;
					st_OUT_PecomMsg.stMsgBuffer[N].MSG[i]	:=	INT_TO_WORD(Puffer.data[k]) ;
				END_FOR;
				st_OUT_PecomMsg.valid[N]	:=	TRUE;
				Puffer.job_running := FALSE;
				Puffer.job_done := TRUE;
				EXIT; 
			ELSE
				N	:=	N + 1;		
			END_IF;
		END_FOR;
	
		Puffer.receiver	:=	Puffer_receiver;
	
		IF		Puffer.job_running
			AND Puffer.data_transfer_ready
		THEN	
			Puffer.job_running := FALSE;
			Puffer.job_done 	:= TRUE;
		END_IF;
	END_IF;

END_IF;

END_FUNCTION_BLOCK

// ---- POUs/Pecom Interface/Pecom_Functions/TCP Msg Handling/Pecom_In_Out_data.TcPOU
PROGRAM Pecom_In_Out_data
VAR
	MAX_ANZ_ZYKL_IN_data_valid:	INT;
	anz_zykl_In_data_valid:	INT;
	ANZBLK_old:	INT;
	ANZBLK:	INT;
	OBJANZ:	INT;
	OBJLGE:	INT;
	i:	INT;
	TON_1:	TON;

END_VAR


(************************************************************************************************)
(*****				 			Pecom In Out Sort subroutine								*****)
(***** If a Pecom Msg contains more the 1 Object... This routine take it					*****) 
(***** apart into single Objects and set the st_IN_Objects.data_are_valid Flag				*****)
(***** until the last object in the message is done											*****)
(************************************************************************************************)

Pecom_In_data();
Pecom_Out_data();
Pecom_Out_Alarm();

ACTION Pecom_In_data:
(*-- Pointer auf naechstes Objekt --*)
IF	st_IN_Objects.data_are_valid
	THEN
		st_IN_Objects.DSK_Pointer 	:= 	st_IN_Objects.DSK_Pointer 
							+ 	OBJLGE;

		IF 		st_IN_Objects.DSK_Pointer > st_IN_Objects.data_Max
			THEN 	
				st_IN_Objects.DSK_Pointer	:= st_IN_Objects.data_Max;
		END_IF;

		IF	OBJANZ <> 0
			THEN (* Bearbeitetes Objekt abziehen *)
				OBJANZ := OBJANZ - 1;
		END_IF;
		
		IF		st_IN_Objects.DSK_Pointer + 2	>=	7
			AND	st_IN_Objects.DSK_Pointer + 2	<=	950
			AND	OBJANZ = 0
			THEN	(* Bearbeiteten Block abziehen *)
				ANZBLK 				:= ANZBLK - 1;
				st_IN_Objects.BLK_Pointer 	:= st_IN_Objects.DSK_Pointer;
				i 					:= st_IN_Objects.DSK_Pointer + 2;
				OBJLGE				:= st_IN_Objects.data[i] / 2;
		
		ELSE	(* ABBRUCH *)
				st_IN_Objects.data_are_valid 		:= 	FALSE;
				st_IN_Objects.data_transfer_ready 	:= 	FALSE;
				anz_zykl_In_data_valid		:=	0;
		END_IF;
		
		(*-- Überprüfung Abarbeitung der IN-data --*)
		IF		ANZBLK_old
			=	ANZBLK	
			THEN
				anz_zykl_In_data_valid	:=	anz_zykl_In_data_valid	+	1;

				IF		anz_zykl_In_data_valid
					>=	MAX_ANZ_ZYKL_IN_data_valid
					THEN
						ANZBLK	:=	0;
				END_IF;
		END_IF;

		ANZBLK_old	:=	ANZBLK;

		(*-- Ende Dekodierung --*)
		IF	ANZBLK = 0
			THEN
				st_IN_Objects.data_are_valid 		:= 	FALSE;
				st_IN_Objects.data_transfer_ready 	:= 	FALSE;
				anz_zykl_In_data_valid		:=	0;	
		END_IF;
END_IF;

(*------------------------------------------------------------------------------------------*)
(*-- Initialisierung --*)
IF 	st_IN_Objects.BLK_Pointer = 0 
	THEN 
		st_IN_Objects.BLK_Pointer := 9; 
END_IF;

IF 	st_IN_Objects.DSK_Pointer = 0 
	THEN 
		st_IN_Objects.DSK_Pointer := 12; 
END_IF;
st_IN_Objects.data_Max := 930;

(*------------------------------------------------------------------------------------------*)
(*-- Start Dekodierung --*)
IF		NOT	st_IN_Objects.data_are_valid
	AND	st_IN_Objects.data_transfer_ready
	THEN
		st_IN_Objects.data_are_valid	:=	TRUE;
		st_IN_Objects.BLK_Pointer 			:= 	9;
		st_IN_Objects.DSK_Pointer 			:= 	9;
		ANZBLK						:= st_IN_Objects.data[8];

		IF 	(*	st_IN_Objects.KDO <>  10921 	// Drive Messages
			AND *)
			(st_IN_Objects.KDO < 10901 
			OR 	st_IN_Objects.KDO > 10912)
			THEN
				ANZBLK := 1;
				OBJANZ := 1;
				OBJLGE := 0;
		END_IF;
END_IF;

IF		(st_IN_Objects.KDO >= 10901
	AND	st_IN_Objects.KDO <= 10912
	OR  st_IN_Objects.KDO =  10921)		// Drive Messages
	AND	st_IN_Objects.BLK_Pointer =	st_IN_Objects.DSK_Pointer
	AND	st_IN_Objects.data_are_valid
	THEN	(* 1. Objekt im Block *)
		IF		st_IN_Objects.DSK_Pointer + 1	>=	7
			AND	st_IN_Objects.DSK_Pointer + 1	<=	950
			AND	st_IN_Objects.DSK_Pointer + 2	>=	7
			AND	st_IN_Objects.DSK_Pointer + 2	<=	950
			THEN
				i 		:= st_IN_Objects.DSK_Pointer + 1;
				OBJANZ	:= st_IN_Objects.data[i];

				i 		:= st_IN_Objects.DSK_Pointer + 2;
				OBJLGE	:= st_IN_Objects.data[i] / 2;

				st_IN_Objects.DSK_Pointer 	:= 
										st_IN_Objects.BLK_Pointer 
									+ 	3;
		
		ELSE	(* ABBRUCH *)
				st_IN_Objects.data_are_valid 		:= 	FALSE;
				st_IN_Objects.data_transfer_ready 	:= 	FALSE;
				anz_zykl_In_data_valid		:=	0;
		END_IF;
END_IF;
END_ACTION

ACTION Pecom_Out_Alarm:
(**********************************************************************************)
(***  Pecom Alarm messages OUT 													***)
(*** the struct "OUT_MSG" is transfered to the send Buffer  "OUT_MSG_puffer"	***)
(**********************************************************************************)
st_OUT_Alarms.Error 					:=	st_OUT_Alarms_Buffer.Error;
st_OUT_Alarms.Hand_Shake				:=	st_OUT_Alarms_Buffer.Hand_Shake;
st_OUT_Alarms.nNumber_of_messages		:=	st_OUT_Alarms_Buffer.nNumber_of_messages;
st_OUT_Alarms.nNumber_of_Error			:=	st_OUT_Alarms_Buffer.nNumber_of_Error;
st_OUT_Alarms.nUnknown_message			:=	st_OUT_Alarms_Buffer.nUnknown_message;
st_OUT_Alarms.data_transfer_ready		:=	st_OUT_Alarms_Buffer.data_transfer_ready;
st_OUT_Alarms.job_running				:=	st_OUT_Alarms_Buffer.job_running;
st_OUT_Alarms.job_done					:=	st_OUT_Alarms_Buffer.job_done;
st_OUT_Alarms.job_not_done				:=	st_OUT_Alarms_Buffer.job_not_done;
st_OUT_Alarms.job_timeout				:=	st_OUT_Alarms_Buffer.job_timeout;

IF		NOT st_OUT_Alarms_Buffer.data_are_valid
	AND NOT st_OUT_Alarms_Buffer.data_transfer_ready
	AND	st_OUT_Alarms.DSK_Pointer > 8
	THEN	
		st_OUT_Alarms.BLK_Pointer := 0; (* number of Alarms *)
		st_OUT_Alarms.DSK_Pointer := 8;

		IF	st_OUT_Alarms.receiver	>	0
			THEN	(* data für Senden *)
				st_OUT_Alarms_Buffer.receiver				:=	st_OUT_Alarms.receiver;
				st_OUT_Alarms_Buffer.Sender					:=	st_OUT_Alarms.Sender;
				st_OUT_Alarms_Buffer.Typ					:=	st_OUT_Alarms.Typ;
				st_OUT_Alarms_Buffer.NFB					:=	st_OUT_Alarms.NFB;
				st_OUT_Alarms_Buffer.Lg_Byte				:=	st_OUT_Alarms.Lg_Byte;
				st_OUT_Alarms_Buffer.KDO					:=	st_OUT_Alarms.KDO;		 
				
				st_OUT_Alarms_Buffer.data 					:=	st_OUT_Alarms.data; 

				st_OUT_Alarms_Buffer.data_are_valid		:=	TRUE;

				st_OUT_Alarms.receiver 					:= 	0;
		END_IF;
END_IF;

IF	(	st_OUT_Alarms_Buffer.job_done
	OR	st_OUT_Alarms_Buffer.job_not_done)
	AND	st_OUT_Alarms_Buffer.data_are_valid
	AND	st_OUT_Alarms_Buffer.data_transfer_ready
	THEN
		st_OUT_Alarms_Buffer.data_are_valid    	:=	FALSE;
		st_OUT_Alarms_Buffer.data_transfer_ready 	:= 	FALSE;
		st_OUT_Alarms_Buffer.receiver 				:= 	0;
END_IF;

IF 	st_OUT_Alarms.DSK_Pointer = 0 
	THEN 
		st_OUT_Alarms.DSK_Pointer := 8; 
END_IF;

st_OUT_Alarms.data_Max := 900;

TON_1 ( IN := NOT st_OUT_Alarms.Release_first_value,
		PT := T#4s); (* release first value bit after 4 sec *)
IF		TON_1.Q
	THEN	
		st_OUT_Alarms.Release_first_value := TRUE;
END_IF;
END_ACTION

ACTION Pecom_Out_data:
(**********************************************************************************)
(***  Pecom Object messages OUT 												***)
(* the struct "OUT_Objects_puffer" is sorted and transfered to -> "OUT_Objects" ***)
(**********************************************************************************)
st_OUT_Objects.Error 						:=	st_OUT_Objects_Buffer.Error;
st_OUT_Objects.Hand_Shake					:=	st_OUT_Objects_Buffer.Hand_Shake;
st_OUT_Objects.nNumber_of_messages			:=	st_OUT_Objects_Buffer.nNumber_of_messages;
st_OUT_Objects.nNumber_of_Error				:=	st_OUT_Objects_Buffer.nNumber_of_Error;
st_OUT_Objects.nUnknown_message				:=	st_OUT_Objects_Buffer.nUnknown_message;
st_OUT_Objects.data_transfer_ready			:=	st_OUT_Objects_Buffer.data_transfer_ready;
st_OUT_Objects.job_running					:=	st_OUT_Objects_Buffer.job_running;
st_OUT_Objects.job_done						:=	st_OUT_Objects_Buffer.job_done;
st_OUT_Objects.job_not_done					:=	st_OUT_Objects_Buffer.job_not_done;
st_OUT_Objects.job_timeout					:=	st_OUT_Objects_Buffer.job_timeout;

IF		NOT st_OUT_Objects_Buffer.data_are_valid
	AND NOT st_OUT_Objects_Buffer.data_transfer_ready
	AND	st_OUT_Objects.DSK_Pointer > 12 
	THEN	
		st_OUT_Objects.BLK_Pointer 					:=	9;
		st_OUT_Objects.DSK_Pointer 					:=	12;

		IF	st_OUT_Objects.receiver	>	0
			THEN	(* data für Senden *)
				st_OUT_Objects_Buffer.receiver		:=	st_OUT_Objects.receiver;
				st_OUT_Objects_Buffer.Typ			:=	st_OUT_Objects.Typ;
				st_OUT_Objects_Buffer.NFB			:=	st_OUT_Objects.NFB;
				st_OUT_Objects_Buffer.Lg_Byte		:=	st_OUT_Objects.Lg_Byte;
				st_OUT_Objects_Buffer.KDO			:=	st_OUT_Objects.KDO;		 
				
				st_OUT_Objects_Buffer.data 			:=	st_OUT_Objects.data; 

				st_OUT_Objects_Buffer.data_are_valid:=	TRUE;
		END_IF;
END_IF;

(*-- Bereichsgrenzen überwachen --*)
(*-- Struktur OUT_Objects --*)
IF 	st_OUT_Objects.BLK_Pointer = 0 
	THEN 
		st_OUT_Objects.BLK_Pointer := 9; 
END_IF;

IF 	st_OUT_Objects.DSK_Pointer = 0 
	THEN 
		st_OUT_Objects.DSK_Pointer := 12; 
END_IF;

st_OUT_Objects.data_Max := 930;

(*-- Struktur OUT_Objects_puffer --*)
IF 	st_OUT_Objects_Buffer.BLK_Pointer = 0 
	THEN 
		st_OUT_Objects_Buffer.BLK_Pointer := 9; 
END_IF;

IF 	st_OUT_Objects_Buffer.DSK_Pointer = 0 
	THEN 
		st_OUT_Objects_Buffer.DSK_Pointer := 12; 
END_IF;

st_OUT_Objects_Buffer.data_Max := 930;
END_ACTION

END_PROGRAM

// ---- POUs/Pecom Interface/PB_Start_UDP.TcPOU
PROGRAM PB_Start_UDP
VAR_INPUT
	iResetUDP_Com		: BOOL;
END_VAR
	
VAR
	IP_UDP_Server		: ARRAY[1..NR_OF_DRIVEMASTERS] OF IP_C;
	FB_UDP_Server		: ARRAY[1..NR_OF_DRIVEMASTERS] OF FB_UDP_Server;	
	S_BUF_UDP			: ARRAY[1..NR_OF_DRIVEMASTERS] OF ST_UDP_Buffer;		// UDP Send Buffer It is hand over to the UDP Socket 
	R_BUF_UDP			: ARRAY[1..NR_OF_DRIVEMASTERS] OF ST_UDP_Buffer;		// UDP Receive Buffer It comes from the UDP Socket


	IP_UDP_Server_1		: IP_C;
	FB_UDP_Server_1		: FB_UDP_Server;	
	S_BUF_UDP_1			: ST_UDP_Buffer;		// UDP Send Buffer It is hand over to the UDP Socket 
	R_BUF_UDP_1			: ST_UDP_Buffer;		// UDP Receive Buffer It comes from the UDP Socket
                          
	IP_UDP_Server_2		: IP_C;
	FB_UDP_Server_2		: FB_UDP_Server;	
	S_BUF_UDP_2			: ST_UDP_Buffer;		// UDP Send Buffer It is hand over to the UDP Socket 
	R_BUF_UDP_2			: ST_UDP_Buffer;		// UDP Receive Buffer It comes from the UDP Socket
	
	
	
	i: INT;
	nCounter: DINT;
END_VAR

(************************************************************************************************)
(*****				 					Ethernet UDP 										*****)
(***** UDP Communication between the PLC <--> Drive System 									*****)
(***** 																						*****)
(************************************************************************************************)

(*
	(***** UDP Server Start Listen 	******)
	IP_UDP_Server_1.C_ENABLE 	:= NOT iResetUDP_Com;	
	FB_UDP_Server_1(PORT		:= WORD#8101,
					sLocal_IP	:= '172.25.9.5',	// Important if you have more ethernet devices on your plc
					TIME_OUT	:= T#10S,
					IP_C		:= IP_UDP_Server_1,				// Ip settings
					S_BUF		:= S_BUF_UDP_1,
					R_BUF		:= R_BUF_UDP_1);
	
	IP_UDP_Server_1.ERROR;
	IP_UDP_Server_1.C_STATE;	
	IP_UDP_Server_1.TIME_RESET	:= iResetUDP_Com;


	FB_UDP_Connection_arr[5](	sRemote_IP		:= stSetup_DriveCom[5].sRemoteIP, 		// '172.25.4.1', 
								nDriveMemberNr	:= stSetup_DriveCom[5].nDriveMemberNr, 	// 2101, 
								nPLCMemberNr	:= stSetup_DriveCom[5].nPLCMemberNr,	// 5001, 
								p_UDP_DriveData	:= ADR(stDrive_Data_arr[5]), 
								S_BUF			:= ADR(S_BUF_UDP_1),
								R_BUF			:= ADR(R_BUF_UDP_1), 
								bAlarmNoConnection=> bAlarm_NoUDP_Connection[5]);

	(***** UDP Server Start Listen 	******)
	IP_UDP_Server_2.C_ENABLE 	:= NOT iResetUDP_Com;	
	FB_UDP_Server_2(PORT		:= WORD#8101,
					sLocal_IP	:= '172.25.9.6',	// Important if you have more ethernet devices on your plc
					TIME_OUT	:= T#10S,
					IP_C		:= IP_UDP_Server_2,				// Ip settings
					S_BUF		:= S_BUF_UDP_2,
					R_BUF		:= R_BUF_UDP_2);
	
	IP_UDP_Server_2.ERROR;
	IP_UDP_Server_2.C_STATE;	
	IP_UDP_Server_2.TIME_RESET	:= iResetUDP_Com;


	FB_UDP_Connection_arr[6](	sRemote_IP		:= stSetup_DriveCom[6].sRemoteIP, 		// '172.25.4.1', 
								nDriveMemberNr	:= stSetup_DriveCom[6].nDriveMemberNr, 	// 2101, 
								nPLCMemberNr	:= stSetup_DriveCom[6].nPLCMemberNr,	// 5001, 
								p_UDP_DriveData	:= ADR(stDrive_Data_arr[6]), 
								S_BUF			:= ADR(S_BUF_UDP_2),
								R_BUF			:= ADR(R_BUF_UDP_2), 
								bAlarmNoConnection=> bAlarm_NoUDP_Connection[6]);
*)

(*************************************)
(***** UDP Server Start Listen 	******)
(*************************************)

FOR i := 1 TO NR_OF_DRIVEMASTERS DO 	
	
	(***** UDP Server Start Listen 	******)
	IP_UDP_Server[i].C_ENABLE 	:= NOT iResetUDP_Com;	
	FB_UDP_Server[i](PORT		:= WORD#8101,
					sLocal_IP	:= stSetup_DriveCom[i].sLocalIP,	// Important if you have more ethernet devices on your plc
					TIME_OUT	:= T#10S,
					IP_C		:= IP_UDP_Server[i],				// Ip settings
					S_BUF		:= S_BUF_UDP[i],
					R_BUF		:= R_BUF_UDP[i]);
	
	IP_UDP_Server[i].ERROR;
	IP_UDP_Server[i].C_STATE;	
	IP_UDP_Server[i].TIME_RESET	:= iResetUDP_Com;
	
	(*** read the Buffer into the UPD Drive array  ***)
	FB_UDP_Connection_arr[i](	sRemote_IP		:= stSetup_DriveCom[i].sRemoteIP, 		// '172.25.4.1', 
								nDriveMemberNr	:= stSetup_DriveCom[i].nDriveMemberNr, 	// 2101, 
								nPLCMemberNr	:= stSetup_DriveCom[i].nPLCMemberNr,	// 5001, 
								p_UDP_DriveData	:= ADR(stDrive_Data_arr[i]), 
								S_BUF			:= ADR(S_BUF_UDP[i]),
								R_BUF			:= ADR(R_BUF_UDP[i]), 
								bAlarmNoConnection=> bAlarm_NoUDP_Connection[i]);
END_FOR

END_PROGRAM

// ---- POUs/Pecom Interface/Pecom_Functions/TCP Msg Handling/Trigger.TcPOU
FUNCTION_BLOCK Trigger
VAR_INPUT
	iTRIG:	BOOL;
END_VAR
VAR_OUTPUT
	Q:	BOOL;
END_VAR
VAR
	R_TRIG_Ein:	R_TRIG;
	R_TRIG_Quit:	R_TRIG;
	F_TRIG_Ein:	F_TRIG;


	F_TRIG_Quit: F_TRIG;
END_VAR

(* Abfrage des Ereignisses auf Flanke und Quittung zur Wiederholung der Meldung *)

R_TRIG_Ein	(CLK := (iTRIG));
F_TRIG_Ein	(CLK := (iTRIG));
//R_TRIG_Quit	(CLK := LS_RW.OBJ65101.Quit_1s);
F_TRIG_Quit	(CLK := stPecomRW.OBJ_RW_65101.Quit_1s  AND iTRIG );

Q := R_TRIG_EIN.Q OR F_TRIG_EIN.Q OR R_TRIG_Quit.Q OR F_TRIG_Quit.Q;

END_FUNCTION_BLOCK

// ---- POUs/Pecom Interface/Pecom_Functions/Pecom_DriveMessage.TcPOU
FUNCTION_BLOCK Pecom_DriveMessage
VAR_INPUT
	Command_Nr		:	INT;
	RemoteMember	:	INT;
	OBJKNG			:	INT;
	OBJART			:	INT;
	OBJGRP			:	INT;
	OBJEIN			:	INT;
	OBJLFN			:	INT;
	OBJLGE			:	INT;
	SNSTIV_MIN		:	INT;
	nDataBlockSize	:	INT;
	Movement_Active	:	BOOL;
	ParameterNr		:	INT;
END_VAR
VAR_OUTPUT
END_VAR
VAR_IN_OUT
	OBJVAR:	ST_Objekt;

END_VAR
VAR
	Old_TLN					:	ARRAY [0..4] OF ARRAY [0..30] OF INT;
	MAX_ANZ_SEKTIONEN		:	INT := 20;
	DEFAULT_LST				:	INT	:=	70;
	DEFAULT_FE				:	INT	:=	2500;
	DEFAULT_WE				:	INT	:=	5300;
	SNSTIV_MAX				:	INT	:=	32767;

	bBit_Change_1			:	INT;
	bBit_Change_2			:	INT;
	ZYKTME_MIN				:	INT	:=	1;
	ZYKTME_MAX				:	INT :=	32767;
	nNumber					:	INT;
	iw_anf					:	INT;
	p_art					:	INT;
	p_anz					:	INT;
	p_lge					:	INT;
	p_grp					:	INT;
	p_ein					:	INT;
	p_lfn					:	INT;
	p_dat					:	INT;
	nMessage_ID				:	INT;	// Kennung
	nCmd_Number				:	INT;	// Kommando Nummer
	nCMD_Type				:	INT;	// Kommando Typ
			
	sens_nr_start			:	INT;
	sens_nr_ende			:	INT;
	ANFTYP					:	INT;	
	SNSTIV					:	INT;
	ZYKTME					:	INT;
	MASEIN					:	INT;
	nDataCounter				:	INT;
	nCounterEnd				:	INT;
	bInserted				:	BOOL;
	delete_TLN				:	ST_Elements;
	zyktme_akt				:	INT;
	obj_cnt					:	INT;
	counter					: 	UINT;
	divisor					:	DINT;
	i						:	INT;
	k						:	INT;
	ntestcount: INT;
	nTestArrayInt			:	ARRAY[0..100] of INT;
END_VAR

(**********************************************************************************)
(***  Pecom Object Handling 													***)
(***  Must be called in the main program like this (eg. Webtension Splicer 110)	***)
(***                                                                            ***)
(*** 	The Variables are defined as:											***)
(*** 	web_tension		: 	ST_Objekt;                                          ***)
(*** 	web_tension_110	:	Pecom_Message;                                      ***)
(***                                                                            ***)
(***  web_tension_110(RemoteMember:=  Config.prod.Zuordnung_zu_LST_Nr,			***)
(***               OBJART      :=  10506,                                       ***)
(***               OBJGRP      :=  110,                                         ***)
(***               OBJEIN      :=  g_stPecomSetup_Machine.RWA_nr,               ***)
(***               OBJLFN      :=  -1,                                          ***)
(***               OBJLGE      :=  12,                                          ***)
(***               OBJVAR      :=  web_tension,                                 ***)
(***               SNSTIV_MIN  :=  0,                                           ***)
(***               );                                                           ***)
(***                                                                            ***)
(**********************************************************************************)

Write_Out_Message();
Read_In_Message();

ACTION Read_In_Message:
(* is a message valid ?-*)

OBJVAR.Read_Data := FALSE;  (* only for one cycle *)

IF NOT st_IN_Objects.data_are_valid
	THEN
	 	RETURN;
END_IF;

(* Pointer  *)
p_art 		:= 	st_IN_Objects.BLK_Pointer;
p_anz 		:= 	st_IN_Objects.BLK_Pointer + 1;
p_lge 		:= 	st_IN_Objects.BLK_Pointer + 2;
p_grp 		:= 	st_IN_Objects.DSK_Pointer;
p_ein 		:= 	st_IN_Objects.DSK_Pointer + 1;
p_lfn 		:= 	st_IN_Objects.DSK_Pointer + 2;		
p_dat 		:= 	st_IN_Objects.DSK_Pointer + 3;	

IF 		st_IN_Objects.KDO =	10921					(* Drive Communication	*)
	AND st_IN_Objects.data[p_grp]		= 	OBJGRP	(* always needed *)
	AND (	st_IN_Objects.data[p_art]	= 	OBJART
		OR 	OBJART = -1)							(* Read All, can be used *)
	AND (	st_IN_Objects.data[p_ein]	= 	OBJEIN
		OR 	OBJEIN = -1)							(* Read All,can be used  *)
	AND (	st_IN_Objects.data[p_lfn]	= 	OBJLFN
		OR 	OBJLFN = -1)							(* Read All,can be used  *)
	AND (	RemoteMember 				= -1 		(* Read All,can be used  *)
		OR 	RemoteMember = 	st_IN_Objects.Sender)
	AND (	ParameterNr = 	st_IN_Objects.data[15])	(* Specify the parameter from Old Baumüller system eg.1680=Handshake 850=Drivecontrol  *)
		
	THEN 
		OBJVAR.OBJART  := st_IN_Objects.data[p_art];
		OBJVAR.OBJLGE  := st_IN_Objects.data[p_lge];
		OBJVAR.OBJGRP  := st_IN_Objects.data[p_grp];
		OBJVAR.OBJEIN  := st_IN_Objects.data[p_ein];
		OBJVAR.OBJLFN  := st_IN_Objects.data[p_lfn];
		OBJVAR.AUFTRAG := INT#0;
		OBJVAR.TLN[0].flag 		:= TRUE;	
		OBJVAR.TLN[0].KNG   	:= st_IN_Objects.data[7];
		OBJVAR.TLN[0].Nummer	:= st_IN_Objects.Sender;
		OBJVAR.Read_Data 		:= TRUE;		 		
		obj_cnt 				:= obj_cnt +1;
	
		IF 	st_IN_Objects.data[p_lge] > 6   				(* look into the message*)
			THEN
				nCounterEnd := (st_IN_Objects.data[p_lge] - INT#6 )/2;

				FOR nDataCounter := 1 TO nCounterEnd DO
					OBJVAR.In_data[nDataCounter] 	:= 	st_IN_Objects.data[p_dat];
					p_dat						:=	p_dat+1;
				END_FOR;
		END_IF;
END_IF;
END_ACTION

ACTION Write_Out_Message:

(* Pointer *)
p_art := st_OUT_Objects.BLK_Pointer;
p_anz := st_OUT_Objects.BLK_Pointer + 1;
p_lge := st_OUT_Objects.BLK_Pointer + 2;
p_grp := st_OUT_Objects.DSK_Pointer;
p_ein := st_OUT_Objects.DSK_Pointer + 1;
p_lfn := st_OUT_Objects.DSK_Pointer + 2;
p_dat := st_OUT_Objects.DSK_Pointer + 3;

IF  	NOT	Movement_Active
	AND	OBJVAR.TLN[0].flag
	AND	OBJVAR.TLN[0].Nummer <> 0
	THEN
		OBJVAR.KOM_RCK 		:=	TRUE;
		iw_anf 				:=	0;
END_IF;

(* build the message*)
IF		st_OUT_Objects.DSK_Pointer = 12
	AND ( 	st_OUT_Objects.DSK_Pointer <  st_OUT_Objects.data_Max - OBJLGE / 2
		AND	OBJLGE > INT#0
		OR	st_OUT_Objects.DSK_Pointer <  st_OUT_Objects.data_Max - nDataBlockSize / 2)
	AND NOT st_OUT_Objects.data_are_valid
	AND	(	OBJVAR.KOM_RCK )
	THEN
		st_OUT_Objects.KDO			:=	10922;
		st_OUT_Objects.receiver 	:=	OBJVAR.TLN[0].Nummer;
		st_OUT_Objects.Sender		:=	0;
		st_OUT_Objects.Typ		  	:=	153;
		st_OUT_Objects.NFB		  	:=	0;
		st_OUT_Objects.data[7] 	:=	OBJVAR.TLN[0].KNG;		(* this is only a number we must give back *)

		st_OUT_Objects.data[8]     := 1; (* ANZBLK *)
		st_OUT_Objects.data[p_art] := 300;
		st_OUT_Objects.data[p_anz] := 1;  (* OBJANZ *)
		st_OUT_Objects.data[p_lge] := OBJLGE;
		st_OUT_Objects.data[p_grp] := 2054;
		st_OUT_Objects.data[p_ein] := OBJVAR.OBJEIN;
		st_OUT_Objects.data[p_lfn] := OBJVAR.OBJLFN;

		FOR nDataCounter := 1 TO ((OBJLGE-6)/2) DO
			st_OUT_Objects.data[p_dat] := OBJVAR.Out_data[nDataCounter];
			p_dat := p_dat+1;
		END_FOR;

	st_OUT_Objects.DSK_Pointer  := st_OUT_Objects.DSK_Pointer + OBJLGE / 2;

	IF 		st_OUT_Objects.KDO = -432
			OR	st_OUT_Objects.KDO = INT#256
	THEN
			st_OUT_Objects.Lg_Byte := INT#2; (* nur KDO *)
	ELSE	
			st_OUT_Objects.Lg_Byte := ( st_OUT_Objects.DSK_Pointer - 6 ) * 2;
	END_IF;

END_IF;

OBJVAR.TLN[iw_anf].flag	:=	FALSE;
OBJVAR.Send_Data 	   	:=	TRUE;
OBJVAR.KOM_RCK			:=	FALSE;
END_ACTION

END_FUNCTION_BLOCK

// ---- POUs/Pecom Interface/Pecom_Functions/Pecom_Write_Alarm.TcPOU
FUNCTION_BLOCK Pecom_Write_Alarm
VAR_INPUT
	iReceiverPecomNr	:	INT;				// Receiver of the Alarm
	iSenderPecomNr		:	INT;				// Receiver of the Alarm
	Frg					:	BOOL;               // Freigabe Meldung
	StQu				:	BOOL;               // Stoe Quit
	Glob				:	BOOL;               // Global : Umschaltung Meldegruppe 1 und 5 nach 11
	Res					:	INT;                // Reserve
	ort1				:	INT;       
	stAlarm				:	ST_Alarm;  
END_VAR
VAR_OUTPUT
	qAlarmSent			:	BOOL;

END_VAR
VAR	
	Grup				:	INT;                        // Gruppe
	Quit				:	INT;                        // Quittierpflicht
	Sper				:	INT;                        // Sperrzustand
	ErNr				:	INT;                        // Ereignisnummer
	ObjNr				:	INT;                        // Objektnummer
	Mldg				:	BOOL;						// Triggerung Meldung
	            		
